		Get.InputField.r_ApparentPhasePower[Phases.L1]:= r_ApparentPower[Phases.L1];
		Get.InputField.r_ApparentPhasePower[Phases.L2]:= r_ApparentPower[Phases.L2];
		Get.InputField.r_ApparentPhasePower[Phases.L3]:= r_ApparentPower[Phases.L3];		
		Get.InputField.r_ApparentPhasePower[Phases.AVG]:= (r_ApparentPower[Phases.L1] + r_ApparentPower[Phases.L2] + r_ApparentPower[Phases.L3]);	
		Get.InputField.r_ApparentPower := r_ApparentPower[Phases.L1]+ r_ApparentPower[Phases.L2] + r_ApparentPower[Phases.L3];
		
		Get.InputField.r_ReactivePhasePower[Phases.L1]:= r_ReactivePower[Phases.L1];
		Get.InputField.r_ReactivePhasePower[Phases.L2]:= r_ReactivePower[Phases.L2];
		Get.InputField.r_ReactivePhasePower[Phases.L3]:= r_ReactivePower[Phases.L3];		
		Get.InputField.r_ReactivePhasePower[Phases.AVG]:= (r_ReactivePower[Phases.L1] + r_ReactivePower[Phases.L2] + r_ReactivePower[Phases.L3]);	
		Get.InputField.r_ReactivePower := r_ReactivePower[Phases.L1]+ r_ReactivePower[Phases.L2] + r_ReactivePower[Phases.L3];
		
		//Energy Consumed                           
		Get.InputField.r_EnergyConsumed		 :=		LINT_TO_REAL(r_ActiveEnergyNegative);	
	                                                
		//Energy Delivered                          
		Get.InputField.r_EnergySupplied :=		LINT_TO_REAL(r_ActiveEnergyPositive);		
	    
		//Powerfactors                                                                 
	    Get.InputField.r_PowerFactor[Phases.L1]:= r_PowerFactor[Phases.L1];
		Get.InputField.r_PowerFactor[Phases.L2]:= r_PowerFactor[Phases.L2];
		Get.InputField.r_PowerFactor[Phases.L3]:= r_PowerFactor[Phases.L3];		
		Get.InputField.r_PowerFactor[Phases.AVG]:= (r_PowerFactor[Phases.L1] + r_PowerFactor[Phases.L2] + r_PowerFactor[Phases.L3])/3;	                                            

		//THD not in EL3443                                                       
		//VoltageUnbalance  not in EL3443   
		
		//EL3443 only gives a boolean for fieldRotation with True meaning right.
		//So false could be none or left. Check voltages before checking rotation.
		IF (Get.InputField.r_LineVoltage[Phases.L1] > 300) AND (Get.InputField.r_LineVoltage[Phases.L2] > 300) AND (Get.InputField.r_LineVoltage[Phases.L3] > 300) THEN
			IF  TotalStatus.bit_GridDirection THEN
				Get.InputField.e_ACrotationStatus := eACRotationState.Right;
			ELSE
				Get.InputField.e_ACrotationStatus := eACRotationState.Left;	
			END_IF
		ELSE
			Get.InputField.e_ACrotationStatus := eACRotationState.None;	
		END_IF
		get.events.b_EL3443Warning := FALSE;
		EL3443FaultCounter := 0;
		
	ELSE
		//faultwarning sets directly if the card states an error.
		//Fault error only sets if the fault remains for a longer period of time.
		get.events.b_EL3443Warning := TRUE;
		EL3443FaultCounter := EL3443FaultCounter +1;
		IF EL3443FaultCounter > 50 THEN
			get.events.b_EL3443Error := TRUE;
		END_IF
	END_IF
END_IF

END_FUNCTION_BLOCK

// ---- POUs/Objects/PowerQualityMonitor/FB_Janitza_UMG801/FB_Janitza.TcPOU
FUNCTION_BLOCK FB_Janitza
VAR_IN_OUT
	get					: ST_PowerMonitor_get;
END_VAR
VAR
	MBRead: FB_MBReadRegs;
	w_MBStartAddress	:	WORD;
	//Set 1 is bigger, as this includes voltage measurements.
	DataBuffer		: 	ARRAY[0..62] OF REAL;
	SecondDataBuffer		: 	ARRAY[0..62] OF REAL;
	tempword	:	dword;	
	temp	:	BOOL;
	UI_Iterator	:	UINT;
	//retrieve new data every 100ms
	GetDataTimer	:	TON := (PT := TIME#100MS);
END_VAR

VAR_INPUT
	ReadData: BOOL;
	b_TNmodeEnable		AT %Q* : BOOL;
END_VAR

VAR
	ast_InputPowerlockData	:	ARRAY[1..2] OF ST_Powerlockdata;
	ast_OutputPowerlockData	:	ARRAY[1..3] OF ST_Powerlockdata;

	StartTransmissionEdge : R_Trig;
	TransmissionDone	:	F_trig;
	
	ui_MBRetryCount	:	uint;
	
	b_busy: BOOL;
	b_CommError: BOOL;
	udi_errid: UDINT;
	udi_cbread: UDINT;
	
	testWord	:	DWORD;
	testWordB	:	WORD;
	testWordC	:	WORD;
END_VAR



//While ReadData is true, initiate data transfer every 100ms;
GetDataTimer(in:= ((NOT GetDataTimer.Q) AND ReadData));

//ReadJanitzaData();
ReadDataSFC();

ACTION aCombineInputData:
IF PowerMeterConfig.b_InputFieldsAvailable THEN
	//Combine shared data from output fields into get struct
	get.InputField.r_Current[Phases.L1] :=	get.InputField.ar_PowerlockCurrents[1][Phases.L1] + 
											get.InputField.ar_PowerlockCurrents[2][Phases.L1];
	
	get.InputField.r_Current[Phases.L2] :=	get.InputField.ar_PowerlockCurrents[1][Phases.L2] + 
											get.InputField.ar_PowerlockCurrents[2][Phases.L2];
	
	get.InputField.r_Current[Phases.L3] :=	get.InputField.ar_PowerlockCurrents[1][Phases.L3] + 
											get.InputField.ar_PowerlockCurrents[2][Phases.L3];			
	
	get.InputField.r_Current[Phases.N] :=	get.InputField.ar_PowerlockCurrents[1][Phases.N] + 
											get.InputField.ar_PowerlockCurrents[2][Phases.N];			
	
	get.InputField.r_Current[Phases.AVG] :=	(get.InputField.r_Current[Phases.L1] + 
											get.InputField.r_Current[Phases.L2] +
											get.InputField.r_Current[Phases.L3])/3;							
	
	Get.InputField.r_ActivePhasePower[Phases.L1]	:=	ast_InputPowerLockData[1].r_ActivePhasePower[Phases.L1] + 
														ast_InputPowerLockData[2].r_ActivePhasePower[Phases.L1];
	
	Get.InputField.r_ActivePhasePower[Phases.L2]	:=	ast_InputPowerLockData[1].r_ActivePhasePower[Phases.L2] + 
														ast_InputPowerLockData[2].r_ActivePhasePower[Phases.L2];
														
	Get.InputField.r_ActivePhasePower[Phases.L3]	:=	ast_InputPowerLockData[1].r_ActivePhasePower[Phases.L3] + 
														ast_InputPowerLockData[2].r_ActivePhasePower[Phases.L3];
														
	Get.InputField.r_ActivePhasePower[Phases.AVG]	:=	ast_InputPowerLockData[1].r_ActivePhasePower[Phases.AVG] + 
														ast_InputPowerLockData[2].r_ActivePhasePower[Phases.AVG];									
	
														
														
	Get.InputField.r_ApparentPhasePower[Phases.L1]	:=	ast_InputPowerLockData[1].r_ApparentPhasePower[Phases.L1] + 
														ast_InputPowerLockData[2].r_ApparentPhasePower[Phases.L1];
	
	Get.InputField.r_ApparentPhasePower[Phases.L2]	:=	ast_InputPowerLockData[1].r_ApparentPhasePower[Phases.L2] + 
														ast_InputPowerLockData[2].r_ApparentPhasePower[Phases.L2];
														
	Get.InputField.r_ApparentPhasePower[Phases.L3]	:=	ast_InputPowerLockData[1].r_ApparentPhasePower[Phases.L3] + 
														ast_InputPowerLockData[2].r_ApparentPhasePower[Phases.L3];
														
	Get.InputField.r_ApparentPhasePower[Phases.AVG]	:=	ast_InputPowerLockData[1].r_ApparentPhasePower[Phases.AVG] + 
														ast_InputPowerLockData[2].r_ApparentPhasePower[Phases.AVG];	

														
														
	Get.InputField.r_ReactivePhasePower[Phases.L1]	:=	ast_InputPowerLockData[1].r_ReactivePhasePower[Phases.L1] + 
														ast_InputPowerLockData[2].r_ReactivePhasePower[Phases.L1];
	
	Get.InputField.r_ReactivePhasePower[Phases.L2]	:=	ast_InputPowerLockData[1].r_ReactivePhasePower[Phases.L2] + 
														ast_InputPowerLockData[2].r_ReactivePhasePower[Phases.L2];
														
	Get.InputField.r_ReactivePhasePower[Phases.L3]	:=	ast_InputPowerLockData[1].r_ReactivePhasePower[Phases.L3] + 
														ast_InputPowerLockData[2].r_ReactivePhasePower[Phases.L3];
														
	Get.InputField.r_ReactivePhasePower[Phases.AVG]	:=	ast_InputPowerLockData[1].r_ReactivePhasePower[Phases.AVG] + 
														ast_InputPowerLockData[2].r_ReactivePhasePower[Phases.AVG];	


										
	Get.InputField.r_ActivePower		:=	ast_InputPowerLockData[1].r_ActivePower + 
											ast_InputPowerLockData[2].r_ActivePower;
	
	Get.InputField.r_ApparentPower		:=	ast_InputPowerLockData[1].r_ApparentPower + 
											ast_InputPowerLockData[2].r_ApparentPower;
											
	Get.InputField.r_ReactivePower		:=	ast_InputPowerLockData[1].r_ReactivePower + 
											ast_InputPowerLockData[2].r_ReactivePower;
	
	Get.InputField.r_EnergyConsumed		:=	ast_InputPowerLockData[1].r_EnergyConsumed + 
											ast_InputPowerLockData[2].r_EnergyConsumed;
	
	Get.InputField.r_EnergySupplied		:=	ast_InputPowerLockData[1].r_EnergySupplied + 
											ast_InputPowerLockData[2].r_EnergySupplied;
	
	get.InputField.r_PowerFactor[Phases.L1] :=		(ast_InputPowerLockData[1].ar_PowerFactor[Phases.L1] + 
													ast_InputPowerLockData[2].ar_PowerFactor[Phases.L1] )/2;	
														
	get.InputField.r_PowerFactor[Phases.L2] :=		(ast_InputPowerLockData[1].ar_PowerFactor[Phases.L2] + 
													ast_InputPowerLockData[2].ar_PowerFactor[Phases.L2])/2;		
	
	get.InputField.r_PowerFactor[Phases.L3] :=		(ast_InputPowerLockData[1].ar_PowerFactor[Phases.L3] + 
													ast_InputPowerLockData[2].ar_PowerFactor[Phases.L3])/2;
	
	get.InputField.r_THD[Phases.L1] 		:=		(ast_InputPowerLockData[1].ar_THD[Phases.L1] + 
													ast_InputPowerLockData[2].ar_THD[Phases.L1])/2;
														
	get.InputField.r_THD[Phases.L2] 		:=		(ast_InputPowerLockData[1].ar_THD[Phases.L2] + 
													ast_InputPowerLockData[2].ar_THD[Phases.L2])/2;	
	
	get.InputField.r_THD[Phases.L3]		 	:=		(ast_InputPowerLockData[1].ar_THD[Phases.L3] + 
													ast_InputPowerLockData[2].ar_THD[Phases.L3])/2;											
	
	get.InputField.r_PowerFactor[Phases.AVG] :=	(get.InputField.r_PowerFactor[Phases.L1] + 
													get.InputField.r_PowerFactor[Phases.L2] + 
													get.InputField.r_PowerFactor[Phases.L3])/3;		
	
	get.InputField.r_THD[Phases.AVG] :=			(get.InputField.r_THD[Phases.L1] + 
													get.InputField.r_THD[Phases.L2] + 
													get.InputField.r_THD[Phases.L3])/3;
end_if
END_ACTION

ACTION aCombineOutputData:

//Combine shared data from output fields into get struct
get.OutputField.r_Current[Phases.L1] :=	get.OutputField.ar_PowerlockCurrents[1][Phases.L1] + 
										get.OutputField.ar_PowerlockCurrents[2][Phases.L1] + 
										get.OutputField.ar_PowerlockCurrents[3][Phases.L1];

get.OutputField.r_Current[Phases.L2] :=	get.OutputField.ar_PowerlockCurrents[1][Phases.L2] + 
										get.OutputField.ar_PowerlockCurrents[2][Phases.L2] + 
										get.OutputField.ar_PowerlockCurrents[3][Phases.L2];

get.OutputField.r_Current[Phases.L3] :=	get.OutputField.ar_PowerlockCurrents[1][Phases.L3] + 
										get.OutputField.ar_PowerlockCurrents[2][Phases.L3] + 
										get.OutputField.ar_PowerlockCurrents[3][Phases.L3];			

get.OutputField.r_Current[Phases.N] :=	get.OutputField.ar_PowerlockCurrents[1][Phases.N] + 
										get.OutputField.ar_PowerlockCurrents[2][Phases.N] + 
										get.OutputField.ar_PowerlockCurrents[3][Phases.N];			

get.OutputField.r_Current[Phases.AVG] :=	(get.OutputField.r_Current[Phases.L1] + 
											get.OutputField.r_Current[Phases.L2] +
											get.OutputField.r_Current[Phases.L3])/3;							

Get.OutputField.r_ActivePhasePower[Phases.L1]	:=	ast_OutputPowerLockData[1].r_ActivePhasePower[Phases.L1] + 
													ast_OutputPowerLockData[2].r_ActivePhasePower[Phases.L1] +
													ast_OutputPowerLockData[3].r_ActivePhasePower[Phases.L1];
	
Get.OutputField.r_ActivePhasePower[Phases.L2]	:=	ast_OutputPowerLockData[1].r_ActivePhasePower[Phases.L2] + 
													ast_OutputPowerLockData[2].r_ActivePhasePower[Phases.L2] +
													ast_OutputPowerLockData[3].r_ActivePhasePower[Phases.L2];
														
Get.OutputField.r_ActivePhasePower[Phases.L3]	:=	ast_OutputPowerLockData[1].r_ActivePhasePower[Phases.L3] + 
													ast_OutputPowerLockData[2].r_ActivePhasePower[Phases.L3] + 
													ast_OutputPowerLockData[3].r_ActivePhasePower[Phases.L3];
														
Get.OutputField.r_ActivePhasePower[Phases.AVG]	:=	ast_OutputPowerLockData[1].r_ActivePhasePower[Phases.AVG] + 
													ast_OutputPowerLockData[2].r_ActivePhasePower[Phases.AVG] +
													ast_OutputPowerLockData[3].r_ActivePhasePower[Phases.AVG];									
	
														
														
Get.OutputField.r_ApparentPhasePower[Phases.L1]	:=	ast_OutputPowerLockData[1].r_ApparentPhasePower[Phases.L1] + 
													ast_OutputPowerLockData[2].r_ApparentPhasePower[Phases.L1] +
													ast_OutputPowerLockData[3].r_ApparentPhasePower[Phases.L1];
	
Get.OutputField.r_ApparentPhasePower[Phases.L2]	:=	ast_OutputPowerLockData[1].r_ApparentPhasePower[Phases.L2] + 
													ast_OutputPowerLockData[2].r_ApparentPhasePower[Phases.L2] +
													ast_OutputPowerLockData[3].r_ApparentPhasePower[Phases.L2];
														
Get.OutputField.r_ApparentPhasePower[Phases.L3]	:=	ast_OutputPowerLockData[1].r_ApparentPhasePower[Phases.L3] + 
													ast_OutputPowerLockData[2].r_ApparentPhasePower[Phases.L3] +
													ast_OutputPowerLockData[3].r_ApparentPhasePower[Phases.L3];
														
Get.OutputField.r_ApparentPhasePower[Phases.AVG]:=	ast_OutputPowerLockData[1].r_ApparentPhasePower[Phases.AVG] + 
													ast_OutputPowerLockData[2].r_ApparentPhasePower[Phases.AVG] +
													ast_OutputPowerLockData[3].r_ApparentPhasePower[Phases.AVG];	
														
													
													
Get.OutputField.r_ReactivePhasePower[Phases.L1]	:=	ast_OutputPowerLockData[1].r_ReactivePhasePower[Phases.L1] + 
													ast_OutputPowerLockData[2].r_ReactivePhasePower[Phases.L1] +
													ast_OutputPowerLockData[3].r_ReactivePhasePower[Phases.L1];	
	
Get.OutputField.r_ReactivePhasePower[Phases.L2]	:=	ast_OutputPowerLockData[1].r_ReactivePhasePower[Phases.L2] + 
													ast_OutputPowerLockData[2].r_ReactivePhasePower[Phases.L2] +
													ast_OutputPowerLockData[3].r_ReactivePhasePower[Phases.L2];	
														
Get.OutputField.r_ReactivePhasePower[Phases.L3]	:=	ast_OutputPowerLockData[1].r_ReactivePhasePower[Phases.L3] + 
													ast_OutputPowerLockData[2].r_ReactivePhasePower[Phases.L3] +
													ast_OutputPowerLockData[3].r_ReactivePhasePower[Phases.L3];	
														
Get.OutputField.r_ReactivePhasePower[Phases.AVG]:=	ast_OutputPowerLockData[1].r_ReactivePhasePower[Phases.AVG] + 
													ast_OutputPowerLockData[2].r_ReactivePhasePower[Phases.AVG] +	
													ast_OutputPowerLockData[3].r_ReactivePhasePower[Phases.AVG];												
											
											
Get.OutputField.r_ActivePower		:=	ast_OutputPowerLockData[1].r_ActivePower + 
										ast_OutputPowerLockData[2].r_ActivePower + 
										ast_OutputPowerLockData[3].r_ActivePower;

Get.OutputField.r_ApparentPower		:=	ast_OutputPowerLockData[1].r_ApparentPower + 
										ast_OutputPowerLockData[2].r_ApparentPower + 
										ast_OutputPowerLockData[3].r_ApparentPower;

Get.OutputField.r_ReactivePower		:=	ast_OutputPowerLockData[1].r_ReactivePower + 
										ast_OutputPowerLockData[2].r_ReactivePower + 
										ast_OutputPowerLockData[3].r_ReactivePower;

Get.OutputField.r_EnergyConsumed	:=	ast_OutputPowerLockData[1].r_EnergyConsumed + 
										ast_OutputPowerLockData[2].r_EnergyConsumed + 
										ast_OutputPowerLockData[3].r_EnergyConsumed;

Get.OutputField.r_EnergySupplied	:=	ast_OutputPowerLockData[1].r_EnergySupplied + 
										ast_OutputPowerLockData[2].r_EnergySupplied + 
										ast_OutputPowerLockData[3].r_EnergySupplied;

//if 3 output fields are available, calculate averages over 3 fields. Otherwise over 2
IF PowerMeterConfig.b_ThirdOutputFieldAvailable THEN
	get.OutputField.r_PowerFactor[Phases.L1] :=		(ast_OutputPowerLockData[1].ar_PowerFactor[Phases.L1] + 
													ast_OutputPowerLockData[2].ar_PowerFactor[Phases.L1] + 
													ast_OutputPowerLockData[3].ar_PowerFactor[Phases.L1])/3;	
													
	get.OutputField.r_PowerFactor[Phases.L2] :=		(ast_OutputPowerLockData[1].ar_PowerFactor[Phases.L2] + 
													ast_OutputPowerLockData[2].ar_PowerFactor[Phases.L2] + 
													ast_OutputPowerLockData[3].ar_PowerFactor[Phases.L2])/3;		

	get.OutputField.r_PowerFactor[Phases.L3] :=		(ast_OutputPowerLockData[1].ar_PowerFactor[Phases.L3] + 
													ast_OutputPowerLockData[2].ar_PowerFactor[Phases.L3] + 
													ast_OutputPowerLockData[3].ar_PowerFactor[Phases.L3])/3;	

	get.OutputField.r_THD[Phases.L1] 		:=		(ast_OutputPowerLockData[1].ar_THD[Phases.L1] + 
													ast_OutputPowerLockData[2].ar_THD[Phases.L1] + 
													ast_OutputPowerLockData[3].ar_THD[Phases.L1])/3;	
													
	get.OutputField.r_THD[Phases.L2] 		:=		(ast_OutputPowerLockData[1].ar_THD[Phases.L2] + 
													ast_OutputPowerLockData[2].ar_THD[Phases.L2] + 
													ast_OutputPowerLockData[3].ar_THD[Phases.L2])/3;		

	get.OutputField.r_THD[Phases.L3]		 :=		(ast_OutputPowerLockData[1].ar_THD[Phases.L3] + 
													ast_OutputPowerLockData[2].ar_THD[Phases.L3] + 
													ast_OutputPowerLockData[3].ar_THD[Phases.L3])/3;														
ELSE
	get.OutputField.r_PowerFactor[Phases.L1] :=		(ast_OutputPowerLockData[1].ar_PowerFactor[Phases.L1] + 
													ast_OutputPowerLockData[2].ar_PowerFactor[Phases.L1] )/2;	
													
	get.OutputField.r_PowerFactor[Phases.L2] :=		(ast_OutputPowerLockData[1].ar_PowerFactor[Phases.L2] + 
													ast_OutputPowerLockData[2].ar_PowerFactor[Phases.L2])/2;		

	get.OutputField.r_PowerFactor[Phases.L3] :=		(ast_OutputPowerLockData[1].ar_PowerFactor[Phases.L3] + 
													ast_OutputPowerLockData[2].ar_PowerFactor[Phases.L3])/2;

	get.OutputField.r_THD[Phases.L1] 		:=		(ast_OutputPowerLockData[1].ar_THD[Phases.L1] + 
													ast_OutputPowerLockData[2].ar_THD[Phases.L1])/2;
													
	get.OutputField.r_THD[Phases.L2] 		:=		(ast_OutputPowerLockData[1].ar_THD[Phases.L2] + 
													ast_OutputPowerLockData[2].ar_THD[Phases.L2])/2;	

	get.OutputField.r_THD[Phases.L3]		 :=		(ast_OutputPowerLockData[1].ar_THD[Phases.L3] + 
													ast_OutputPowerLockData[2].ar_THD[Phases.L3])/2;											
END_IF



get.OutputField.r_PowerFactor[Phases.AVG] :=	(get.OutputField.r_PowerFactor[Phases.L1] + 
												get.OutputField.r_PowerFactor[Phases.L2] + 
												get.OutputField.r_PowerFactor[Phases.L3])/3;		

get.OutputField.r_THD[Phases.AVG] :=			(get.OutputField.r_THD[Phases.L1] + 
												get.OutputField.r_THD[Phases.L2] + 
												get.OutputField.r_THD[Phases.L3])/3;
END_ACTION

ACTION aReadInputField1:

IF NOT PowerMeterConfig.b_InputFieldsAvailable THEN
	//skip this step if input fields are not in use
	SFCTip := TRUE;
ELSE
	
	IF PowerMeterconfig.b_ThirdOutputFieldAvailable THEN
		//if third output field is available, Input field is connected to module 2, so inputfield 1 is address 19600
		w_MBStartAddress := 19600;
	ELSE
		//if no third output field is available, Input field is connected to module 1, so inputfield 1 is address 19400
		w_MBStartAddress := 19400;
	END_IF

	MBRead(
	sIPAddr := PowerMeterConfig.IP_JANITZA,
	nTCPPort := PowerMeterConfig.MBPort_Janitza,
	nUnitID := 1,//16#FF;
	nMBAddr := w_MBStartAddress,
	nQuantity := 50*2,
	cbLength := SIZEOF(DataBuffer),
	pDestAddr := ADR(DataBuffer),
	bExecute := NOT (b_busy OR TransmissionDone.Q),	//	<- werkt dit niet gewoon?
	bBusy => b_busy,
	bError => b_CommError,
	nErrId => udi_errid,
	cbRead => udi_cbread,
	tTimeout := T#25MS
	);
	
	TransmissionDone(clk := b_busy);
	
	IF TransmissionDone.q THEN
		IF NOT b_CommError  THEN	
			
			FOR UI_Iterator := 0 TO 50 BY 1 DO
				DataBuffer[UI_Iterator] := ChangeRealEndianess(DataBuffer[UI_Iterator]);
			END_FOR 
			//field specific data, keep separate at first. Then combine data into get struct in a later step.
			get.InputField.ar_PowerlockCurrents[1][Phases.L1] := DataBuffer[0];
			get.InputField.ar_PowerlockCurrents[1][Phases.L2] := DataBuffer[1];
			get.InputField.ar_PowerlockCurrents[1][Phases.L3] := DataBuffer[2];
			get.InputField.ar_PowerlockCurrents[1][Phases.N] := DataBuffer[3];
			
			ast_InputPowerLockData[1].r_ActivePhasePower[phases.L1] := DataBuffer[4];
       		ast_InputPowerLockData[1].r_ActivePhasePower[phases.L2] := DataBuffer[5];
			ast_InputPowerLockData[1].r_ActivePhasePower[phases.L3] := DataBuffer[6];
			ast_InputPowerLockData[1].r_ActivePhasePower[phases.AVG] := (DataBuffer[4] + DataBuffer[5] + DataBuffer[6])/3;
		    
			ast_InputPowerLockData[1].r_ApparentPhasePower[phases.L1] := DataBuffer[8];
       		ast_InputPowerLockData[1].r_ApparentPhasePower[phases.L2] := DataBuffer[9];
			ast_InputPowerLockData[1].r_ApparentPhasePower[phases.L3] := DataBuffer[10];
			ast_InputPowerLockData[1].r_ApparentPhasePower[phases.AVG] := (DataBuffer[8] + DataBuffer[9] + DataBuffer[10])/3;
		    
			ast_InputPowerLockData[1].r_ReactivePhasePower[phases.L1] := DataBuffer[12];
       		ast_InputPowerLockData[1].r_ReactivePhasePower[phases.L2] := DataBuffer[13];
			ast_InputPowerLockData[1].r_ReactivePhasePower[phases.L3] := DataBuffer[14];
			ast_InputPowerLockData[1].r_ReactivePhasePower[phases.AVG] := (DataBuffer[12] + DataBuffer[13] + DataBuffer[14])/3;
		    
			ast_InputPowerLockData[1].r_ActivePower := DataBuffer[7];
			ast_InputPowerLockData[1].r_ApparentPower := DataBuffer[11];
			ast_InputPowerLockData[1].r_ReactivePower := DataBuffer[15];
					               
			ast_InputPowerLockData[1].ar_PowerFactor[Phases.L1] := DataBuffer[16];
			ast_InputPowerLockData[1].ar_PowerFactor[Phases.L2] := DataBuffer[17];
			ast_InputPowerLockData[1].ar_PowerFactor[Phases.L3] := DataBuffer[18];
			ast_InputPowerLockData[1].ar_PowerFactor[Phases.AVG] := (DataBuffer[16] + DataBuffer[17] + DataBuffer[18])/3;
					               
			ast_InputPowerLockData[1].r_EnergyConsumed	:=  DataBuffer[26];
			ast_InputPowerLockData[1].r_EnergySupplied 	:=	DataBuffer[30];
					               
			ast_InputPowerLockData[1].ar_THD[Phases.L1] := DataBuffer[47];
			ast_InputPowerLockData[1].ar_THD[Phases.L2] := DataBuffer[48];
			ast_InputPowerLockData[1].ar_THD[Phases.L3] := DataBuffer[49];
				
			ui_MBRetryCount := 0;
			sfctip := TRUE;
		ELSE
			ui_MBRetryCount := ui_MBRetryCount + 1;
			
			IF ui_MBRetryCount > 1 THEN
				get.events.b_MBCommWarning := TRUE;
			END_IF	
			
			//if comm fails 5 times in a row. try next input
			IF ui_MBRetryCount > 4 THEN
				get.Events.b_MBCommError := TRUE;
				sfctip := TRUE;
			END_IF
		END_IF
	END_IF
END_IF
END_ACTION

ACTION aReadInputField2:

IF NOT PowerMeterConfig.b_InputFieldsAvailable THEN
	//skip this step if input fields are not in use
	SFCTip := TRUE;
ELSE
	
	IF PowerMeterconfig.b_ThirdOutputFieldAvailable THEN
		//if third output field is available, Input field is connected to module 2, so inputfield 2 is address 19700
		w_MBStartAddress := 19700;
	ELSE
		//if no third output field is available, Input field is connected to module 1, so inputfield 2 is address 19500
		w_MBStartAddress := 19500;
	END_IF

	MBRead(
	sIPAddr := PowerMeterConfig.IP_JANITZA,
	nTCPPort := PowerMeterConfig.MBPort_Janitza,
	nUnitID := 1,//16#FF;
	nMBAddr := w_MBStartAddress,
	nQuantity := 50*2,
	cbLength := SIZEOF(DataBuffer),
	pDestAddr := ADR(DataBuffer),
	bExecute := NOT (b_busy OR TransmissionDone.Q),	//	<- werkt dit niet gewoon?
	bBusy => b_busy,
	bError => b_CommError,
	nErrId => udi_errid,
	cbRead => udi_cbread,
	tTimeout := T#25MS
	);
	
	TransmissionDone(clk := b_busy);
	
	IF TransmissionDone.q THEN
		IF NOT b_CommError THEN	
			
			FOR UI_Iterator := 0 TO 50 BY 1 DO
				DataBuffer[UI_Iterator] := ChangeRealEndianess(DataBuffer[UI_Iterator]);
			END_FOR 
			
			//field specific data, keep separate at first. Then combine data into get struct in a later step.
			get.InputField.ar_PowerlockCurrents[2][Phases.L1] := DataBuffer[0];
			get.InputField.ar_PowerlockCurrents[2][Phases.L2] := DataBuffer[1];
			get.InputField.ar_PowerlockCurrents[2][Phases.L3] := DataBuffer[2];
			get.InputField.ar_PowerlockCurrents[2][Phases.N] := DataBuffer[3];
			
			ast_InputPowerLockData[2].r_ActivePhasePower[phases.L1] := DataBuffer[4];
       		ast_InputPowerLockData[2].r_ActivePhasePower[phases.L2] := DataBuffer[5];
			ast_InputPowerLockData[2].r_ActivePhasePower[phases.L3] := DataBuffer[6];
			ast_InputPowerLockData[2].r_ActivePhasePower[phases.AVG] := (DataBuffer[4] + DataBuffer[5] + DataBuffer[6])/3;
		                           
			ast_InputPowerLockData[2].r_ApparentPhasePower[phases.L1] := DataBuffer[8];
       		ast_InputPowerLockData[2].r_ApparentPhasePower[phases.L2] := DataBuffer[9];
			ast_InputPowerLockData[2].r_ApparentPhasePower[phases.L3] := DataBuffer[10];
			ast_InputPowerLockData[2].r_ApparentPhasePower[phases.AVG] := (DataBuffer[8] + DataBuffer[9] + DataBuffer[10])/3;
		                           
			ast_InputPowerLockData[2].r_ReactivePhasePower[phases.L1] := DataBuffer[12];
       		ast_InputPowerLockData[2].r_ReactivePhasePower[phases.L2] := DataBuffer[13];
			ast_InputPowerLockData[2].r_ReactivePhasePower[phases.L3] := DataBuffer[14];
			ast_InputPowerLockData[2].r_ReactivePhasePower[phases.AVG] := (DataBuffer[12] + DataBuffer[13] + DataBuffer[14])/3;
		    			
			ast_InputPowerLockData[2].r_ActivePower := DataBuffer[7];
			ast_InputPowerLockData[2].r_ApparentPower := DataBuffer[11];
			ast_InputPowerLockData[2].r_ReactivePower := DataBuffer[15];
					               
			ast_InputPowerLockData[2].ar_PowerFactor[Phases.L1] := DataBuffer[16];
			ast_InputPowerLockData[2].ar_PowerFactor[Phases.L2] := DataBuffer[17];
			ast_InputPowerLockData[2].ar_PowerFactor[Phases.L3] := DataBuffer[18];
			ast_InputPowerLockData[2].ar_PowerFactor[Phases.AVG] := (DataBuffer[16] + DataBuffer[17] + DataBuffer[18])/3;
					               
			ast_InputPowerLockData[2].r_EnergyConsumed	:=  DataBuffer[26];
			ast_InputPowerLockData[2].r_EnergySupplied 	:=	DataBuffer[30];
					               
			ast_InputPowerLockData[2].ar_THD[Phases.L1] := DataBuffer[47];
			ast_InputPowerLockData[2].ar_THD[Phases.L2] := DataBuffer[48];
			ast_InputPowerLockData[2].ar_THD[Phases.L3] := DataBuffer[49];
				
			ui_MBRetryCount := 0;
			sfctip := TRUE;
		ELSE
			ui_MBRetryCount := ui_MBRetryCount + 1;
			
			
			IF ui_MBRetryCount > 1 THEN
				get.events.b_MBCommWarning := TRUE;
			END_IF	
			
			//if comm fails 5 times in a row. try next input
			IF ui_MBRetryCount > 4 THEN
				get.Events.b_MBCommError := TRUE;
				sfctip := TRUE;
			END_IF
		END_IF
	END_IF
END_IF
END_ACTION

ACTION aReadInternalField:

MBRead(
sIPAddr := PowerMeterConfig.IP_JANITZA,
nTCPPort := PowerMeterConfig.MBPort_Janitza,
nUnitID := 1,//16#FF;
nMBAddr := 19300,
nQuantity := 50*2,
cbLength := SIZEOF(DataBuffer),
pDestAddr := ADR(DataBuffer),
bExecute := NOT (b_busy OR TransmissionDone.Q),	//	<- werkt dit niet gewoon?
bBusy => b_busy,
bError => b_CommError,
nErrId => udi_errid,
cbRead => udi_cbread,
tTimeout := T#25MS
);

TransmissionDone(clk := b_busy);

IF TransmissionDone.q THEN
	IF NOT b_CommError  THEN	
		
		FOR UI_Iterator := 0 TO 50 BY 1 DO
			DataBuffer[UI_Iterator] := ChangeRealEndianess(DataBuffer[UI_Iterator]);
		END_FOR 
		
		//field specific data, keep separate at first. Then combine data into get struct in a later step.
		get.InternalSupply.r_Current[Phases.L1] := DataBuffer[0];
		get.InternalSupply.r_Current[Phases.L2] := DataBuffer[1];
		get.InternalSupply.r_Current[Phases.L3] := DataBuffer[2];
		get.InternalSupply.r_Current[Phases.N] := DataBuffer[3];
		get.InternalSupply.r_Current[Phases.AVG] := (DataBuffer[0] + DataBuffer[1] + DataBuffer[2])/3;
		
		get.InternalSupply.r_ActivePhasePower[phases.L1] := DataBuffer[4];
   		get.InternalSupply.r_ActivePhasePower[phases.L2] := DataBuffer[5];
		get.InternalSupply.r_ActivePhasePower[phases.L3] := DataBuffer[6];
		get.InternalSupply.r_ActivePhasePower[phases.AVG] := (DataBuffer[4] + DataBuffer[5] + DataBuffer[6])/3;
		
		get.InternalSupply.r_ApparentPhasePower[phases.L1] := DataBuffer[8];
   		get.InternalSupply.r_ApparentPhasePower[phases.L2] := DataBuffer[9];
		get.InternalSupply.r_ApparentPhasePower[phases.L3] := DataBuffer[10];
		get.InternalSupply.r_ApparentPhasePower[phases.AVG] := (DataBuffer[8] + DataBuffer[9] + DataBuffer[10])/3;
		
		get.InternalSupply.r_ReactivePhasePower[phases.L1] := DataBuffer[12];
   		get.InternalSupply.r_ReactivePhasePower[phases.L2] := DataBuffer[13];
		get.InternalSupply.r_ReactivePhasePower[phases.L3] := DataBuffer[14];
		get.InternalSupply.r_ReactivePhasePower[phases.AVG] := (DataBuffer[12] + DataBuffer[13] + DataBuffer[14])/3;
		    				                        
		get.InternalSupply.r_ActivePower := DataBuffer[7];
		get.InternalSupply.r_ApparentPower := DataBuffer[11];
		get.InternalSupply.r_ReactivePower := DataBuffer[15];
        
		get.InternalSupply.r_PowerFactor[Phases.L1] := DataBuffer[16];
		get.InternalSupply.r_PowerFactor[Phases.L2] := DataBuffer[17];
		get.InternalSupply.r_PowerFactor[Phases.L3] := DataBuffer[18];
		get.InternalSupply.r_PowerFactor[Phases.AVG] := (DataBuffer[16] + DataBuffer[17] + DataBuffer[18])/3;
		
		get.InternalSupply.r_EnergyConsumed	:=  DataBuffer[26];
		get.InternalSupply.r_EnergySupplied 	:=	DataBuffer[30];
		
		get.InternalSupply.r_THD[Phases.L1] := DataBuffer[47];
		get.InternalSupply.r_THD[Phases.L2] := DataBuffer[48];
		get.InternalSupply.r_THD[Phases.L3] := DataBuffer[49];
			
		ui_MBRetryCount := 0;
		sfctip := TRUE;
	ELSE
		ui_MBRetryCount := ui_MBRetryCount + 1;
				
		IF ui_MBRetryCount > 1 THEN
			get.events.b_MBCommWarning := TRUE;
		END_IF	
		
		//if comm fails 5 times in a row. try next input
		IF ui_MBRetryCount > 4 THEN
			get.Events.b_MBCommError := TRUE;
			sfctip := TRUE;
		END_IF
	END_IF
END_IF
END_ACTION

ACTION aReadOutputField1:

MBRead(
sIPAddr := PowerMeterConfig.IP_JANITZA,
nTCPPort := PowerMeterConfig.MBPort_Janitza,
nUnitID := 1,
nMBAddr := 19000,
nQuantity := 61*2,
cbLength := SIZEOF(DataBuffer),
pDestAddr := ADR(DataBuffer),
bExecute := NOT (b_busy OR TransmissionDone.Q),	//	<- werkt dit niet gewoon?
bBusy => b_busy,
bError => b_CommError,
nErrId => udi_errid,
cbRead => udi_cbread,
tTimeout := T#25MS
);

TransmissionDone(clk := b_busy);

IF TransmissionDone.q THEN
	Temp := FALSE;
	IF NOT b_CommError then
		//General inputfield data, can be pushed to get struct immediately
		
		FOR UI_Iterator := 0 TO 61 BY 1 DO
			DataBuffer[UI_Iterator] := ChangeRealEndianess(DataBuffer[UI_Iterator]);
		END_FOR 
		
		get.OutputField.r_PhaseVoltage[Phases.L1] := DataBuffer[0];
		get.OutputField.r_PhaseVoltage[Phases.L2] := DataBuffer[1];
		get.OutputField.r_PhaseVoltage[Phases.L3] := DataBuffer[2];
		get.OutputField.r_PhaseVoltage[Phases.AVG] := (DataBuffer[0]+DataBuffer[1]+DataBuffer[2])/3;
		
		get.OutputField.r_LineVoltage[Phases.L1] := DataBuffer[3];
		get.OutputField.r_LineVoltage[Phases.L2] := DataBuffer[4];
		get.OutputField.r_LineVoltage[Phases.L3] := DataBuffer[5];
		get.OutputField.r_LineVoltage[Phases.AVG] := (DataBuffer[3]+DataBuffer[4]+DataBuffer[5])/3;
		
		get.OutputField.r_Frequency	:= DataBuffer[25];
		
		CASE REAL_TO_INT(DataBuffer[26]) OF
			-1 	:	get.OutputField.e_ACrotationStatus := eACRotationState.Left;
			1	:	get.OutputField.e_ACrotationStatus := eACRotationState.Right;
			0	:	get.OutputField.e_ACrotationStatus := eACRotationState.None;
		END_CASE

		//field specific data, keep separate at first. Then combine data into get struct in a later step.
		get.OutputField.ar_PowerlockCurrents[1][Phases.L1] := DataBuffer[6];
		get.OutputField.ar_PowerlockCurrents[1][Phases.L2] := DataBuffer[7];
		get.OutputField.ar_PowerlockCurrents[1][Phases.L3] := DataBuffer[8];
		get.OutputField.ar_PowerlockCurrents[1][Phases.N] := DataBuffer[9];
		
		ast_OutputPowerLockData[1].r_ActivePhasePower[phases.L1] := DataBuffer[10];
   		ast_OutputPowerLockData[1].r_ActivePhasePower[phases.L2] := DataBuffer[11];
		ast_OutputPowerLockData[1].r_ActivePhasePower[phases.L3] := DataBuffer[12];
		ast_OutputPowerLockData[1].r_ActivePhasePower[phases.AVG] := (DataBuffer[10] + DataBuffer[11] + DataBuffer[12])/3;
		                        
		ast_OutputPowerLockData[1].r_ApparentPhasePower[phases.L1] := DataBuffer[14];
   		ast_OutputPowerLockData[1].r_ApparentPhasePower[phases.L2] := DataBuffer[15];
		ast_OutputPowerLockData[1].r_ApparentPhasePower[phases.L3] := DataBuffer[16];
		ast_OutputPowerLockData[1].r_ApparentPhasePower[phases.AVG] := (DataBuffer[14] + DataBuffer[15] + DataBuffer[16])/3;
		                        
		ast_OutputPowerLockData[1].r_ReactivePhasePower[phases.L1] := DataBuffer[18];
   		ast_OutputPowerLockData[1].r_ReactivePhasePower[phases.L2] := DataBuffer[19];
		ast_OutputPowerLockData[1].r_ReactivePhasePower[phases.L3] := DataBuffer[20];
		ast_OutputPowerLockData[1].r_ReactivePhasePower[phases.AVG] := (DataBuffer[18] + DataBuffer[19] + DataBuffer[20])/3;
		    				                        
		ast_OutputPowerLockData[1].r_ActivePower := DataBuffer[13];
		ast_OutputPowerLockData[1].r_ApparentPower := DataBuffer[17];
		ast_OutputPowerLockData[1].r_ReactivePower := DataBuffer[21];

		ast_OutputPowerLockData[1].ar_PowerFactor[Phases.L1] := DataBuffer[22];
		ast_OutputPowerLockData[1].ar_PowerFactor[Phases.L2] := DataBuffer[23];
		ast_OutputPowerLockData[1].ar_PowerFactor[Phases.L3] := DataBuffer[24];
		ast_OutputPowerLockData[1].ar_PowerFactor[Phases.AVG] := (DataBuffer[22] + DataBuffer[23] + DataBuffer[24])/3;
		
		ast_OutputPowerLockData[1].r_EnergyConsumed	:=  DataBuffer[34];
		ast_OutputPowerLockData[1].r_EnergySupplied 	:=	DataBuffer[38];

		ast_OutputPowerLockData[1].ar_THD[Phases.L1] := DataBuffer[58];
		ast_OutputPowerLockData[1].ar_THD[Phases.L2] := DataBuffer[59];
		ast_OutputPowerLockData[1].ar_THD[Phases.L3] := DataBuffer[60];
			
		ui_MBRetryCount := 0;
		sfctip := TRUE;
	ELSE
		ui_MBRetryCount := ui_MBRetryCount + 1;
		
		IF ui_MBRetryCount > 1 THEN
			get.events.b_MBCommWarning := TRUE;
		END_IF	
		
		//if comm fails 5 times in a row. try next input
		IF ui_MBRetryCount > 4 THEN
			get.Events.b_MBCommError := TRUE;
			sfctip := TRUE;
		END_IF
	END_IF
END_IF
END_ACTION

ACTION aReadOutputField2:

MBRead(
sIPAddr := PowerMeterConfig.IP_JANITZA,
nTCPPort := PowerMeterConfig.MBPort_Janitza,
nUnitID := 1,//16#FF,
nMBAddr := 19200,
nQuantity := 50*2,
cbLength := SIZEOF(DataBuffer),
pDestAddr := ADR(DataBuffer),
bExecute := NOT (b_busy OR TransmissionDone.Q),	//	<- werkt dit niet gewoon?
bBusy => b_busy,
bError => b_CommError,
nErrId => udi_errid,
cbRead => udi_cbread,
tTimeout := T#25MS
);

TransmissionDone(clk := b_busy);

IF TransmissionDone.q THEN
	IF NOT b_CommError THEN	
		
		FOR UI_Iterator := 0 TO 50 BY 1 DO
			DataBuffer[UI_Iterator] := ChangeRealEndianess(DataBuffer[UI_Iterator]);
		END_FOR 	
	
		get.OutputField.ar_PowerlockCurrents[2][Phases.L1] := DataBuffer[0];
		get.OutputField.ar_PowerlockCurrents[2][Phases.L2] := DataBuffer[1];
		get.OutputField.ar_PowerlockCurrents[2][Phases.L3] := DataBuffer[2];
		get.OutputField.ar_PowerlockCurrents[2][Phases.N] := DataBuffer[3];

		ast_OutputPowerLockData[2].r_ActivePhasePower[phases.L1] := DataBuffer[4];
   		ast_OutputPowerLockData[2].r_ActivePhasePower[phases.L2] := DataBuffer[5];
		ast_OutputPowerLockData[2].r_ActivePhasePower[phases.L3] := DataBuffer[6];
		ast_OutputPowerLockData[2].r_ActivePhasePower[phases.AVG] := (DataBuffer[4] + DataBuffer[5] + DataBuffer[6])/3;
		
		ast_OutputPowerLockData[2].r_ApparentPhasePower[phases.L1] := DataBuffer[8];
   		ast_OutputPowerLockData[2].r_ApparentPhasePower[phases.L2] := DataBuffer[9];
		ast_OutputPowerLockData[2].r_ApparentPhasePower[phases.L3] := DataBuffer[10];
		ast_OutputPowerLockData[2].r_ApparentPhasePower[phases.AVG] := (DataBuffer[8] + DataBuffer[9] + DataBuffer[10])/3;
		
		ast_OutputPowerLockData[2].r_ReactivePhasePower[phases.L1] := DataBuffer[12];
   		ast_OutputPowerLockData[2].r_ReactivePhasePower[phases.L2] := DataBuffer[13];
		ast_OutputPowerLockData[2].r_ReactivePhasePower[phases.L3] := DataBuffer[14];
		ast_OutputPowerLockData[2].r_ReactivePhasePower[phases.AVG] := (DataBuffer[12] + DataBuffer[13] + DataBuffer[14])/3;
		    				                        
		ast_OutputPowerLockData[2].r_ActivePower := DataBuffer[7];
		ast_OutputPowerLockData[2].r_ApparentPower := DataBuffer[11];
		ast_OutputPowerLockData[2].r_ReactivePower := DataBuffer[15];
                                
		ast_OutputPowerLockData[2].ar_PowerFactor[Phases.L1] := DataBuffer[16];
		ast_OutputPowerLockData[2].ar_PowerFactor[Phases.L2] := DataBuffer[17];
		ast_OutputPowerLockData[2].ar_PowerFactor[Phases.L3] := DataBuffer[18];
		ast_OutputPowerLockData[2].ar_PowerFactor[Phases.AVG] := (DataBuffer[16] + DataBuffer[17] + DataBuffer[18])/3;
		                        
		ast_OutputPowerLockData[2].r_EnergyConsumed	:=  DataBuffer[26];
		ast_OutputPowerLockData[2].r_EnergySupplied 	:=	DataBuffer[30];
				                
		ast_OutputPowerLockData[2].ar_THD[Phases.L1] := DataBuffer[47];
		ast_OutputPowerLockData[2].ar_THD[Phases.L2] := DataBuffer[48];
		ast_OutputPowerLockData[2].ar_THD[Phases.L3] := DataBuffer[49];
			
		ui_MBRetryCount := 0;
		sfctip := TRUE;
	ELSE
		ui_MBRetryCount := ui_MBRetryCount + 1;
		
		IF ui_MBRetryCount > 1 THEN
			get.events.b_MBCommWarning := TRUE;
		END_IF	
		
		//if comm fails 5 times in a row. try next input
		IF ui_MBRetryCount > 4 THEN
			get.Events.b_MBCommError := TRUE;
			sfctip := TRUE;
		END_IF
	END_IF
END_IF
END_ACTION

ACTION aReadOutputField3:

IF NOT PowerMeterConfig.b_ThirdOutputFieldAvailable THEN
	//skip this step if third field isn't in use
	SFCTip := TRUE;
ELSE
	MBRead(
	sIPAddr := PowerMeterConfig.IP_JANITZA,
	nTCPPort := PowerMeterConfig.MBPort_Janitza,
	nUnitID := 1,//16#FF;
	nMBAddr := 19400,
	nQuantity := 50*2,
	cbLength := SIZEOF(SecondDataBuffer),
	pDestAddr := ADR(SecondDataBuffer),
	bExecute := NOT (b_busy OR TransmissionDone.Q),	//	<- werkt dit niet gewoon?
	bBusy => b_busy,
	bError => b_CommError,
	nErrId => udi_errid,
	cbRead => udi_cbread,
	tTimeout := T#25MS
	);
	
	TransmissionDone(clk := b_busy);
	
	IF TransmissionDone.q THEN
		IF NOT b_CommError  THEN	
			
			FOR UI_Iterator := 0 TO 50 BY 1 DO
				DataBuffer[UI_Iterator] := ChangeRealEndianess(SecondDataBuffer[UI_Iterator]);
			END_FOR 
			//field specific data, keep separate at first. Then combine data into get struct in a later step.
			get.OutputField.ar_PowerlockCurrents[3][Phases.L1] := DataBuffer[0];
			get.OutputField.ar_PowerlockCurrents[3][Phases.L2] := DataBuffer[1];
			get.OutputField.ar_PowerlockCurrents[3][Phases.L3] := DataBuffer[2];
			get.OutputField.ar_PowerlockCurrents[3][Phases.N] := DataBuffer[3];

			ast_OutputPowerLockData[3].r_ActivePhasePower[phases.L1] := DataBuffer[4];
 	  		ast_OutputPowerLockData[3].r_ActivePhasePower[phases.L2] := DataBuffer[5];
			ast_OutputPowerLockData[3].r_ActivePhasePower[phases.L3] := DataBuffer[6];
			ast_OutputPowerLockData[3].r_ActivePhasePower[phases.AVG] := (DataBuffer[4] + DataBuffer[5] + DataBuffer[6])/3;
		                            
			ast_OutputPowerLockData[3].r_ApparentPhasePower[phases.L1] := DataBuffer[8];
	   		ast_OutputPowerLockData[3].r_ApparentPhasePower[phases.L2] := DataBuffer[9];
			ast_OutputPowerLockData[3].r_ApparentPhasePower[phases.L3] := DataBuffer[10];
			ast_OutputPowerLockData[3].r_ApparentPhasePower[phases.AVG] := (DataBuffer[8] + DataBuffer[9] + DataBuffer[10])/3;
		                            
			ast_OutputPowerLockData[3].r_ReactivePhasePower[phases.L1] := DataBuffer[12];
 	 		ast_OutputPowerLockData[3].r_ReactivePhasePower[phases.L2] := DataBuffer[13];
			ast_OutputPowerLockData[3].r_ReactivePhasePower[phases.L3] := DataBuffer[14];
			ast_OutputPowerLockData[3].r_ReactivePhasePower[phases.AVG] := (DataBuffer[12] + DataBuffer[13] + DataBuffer[14])/3;
		    				                        
			ast_OutputPowerLockData[3].r_ActivePower := DataBuffer[7];
			ast_OutputPowerLockData[3].r_ApparentPower := DataBuffer[11];
			ast_OutputPowerLockData[3].r_ReactivePower := DataBuffer[15];
									
			ast_OutputPowerLockData[3].ar_PowerFactor[Phases.L1] := DataBuffer[16];
			ast_OutputPowerLockData[3].ar_PowerFactor[Phases.L2] := DataBuffer[17];
			ast_OutputPowerLockData[3].ar_PowerFactor[Phases.L3] := DataBuffer[18];
			ast_OutputPowerLockData[3].ar_PowerFactor[Phases.AVG] := (DataBuffer[16] + DataBuffer[17] + DataBuffer[18])/3;
									
			ast_OutputPowerLockData[3].r_EnergyConsumed	:=  DataBuffer[26];
			ast_OutputPowerLockData[3].r_EnergySupplied 	:=	DataBuffer[30];
									
			ast_OutputPowerLockData[3].ar_THD[Phases.L1] := DataBuffer[47];
			ast_OutputPowerLockData[3].ar_THD[Phases.L2] := DataBuffer[48];
			ast_OutputPowerLockData[3].ar_THD[Phases.L3] := DataBuffer[49];
				
			ui_MBRetryCount := 0;
			sfctip := TRUE;
		ELSE
			ui_MBRetryCount := ui_MBRetryCount + 1;

			IF ui_MBRetryCount > 1 THEN
				get.events.b_MBCommWarning := TRUE;
			END_IF	
			
			//if comm fails 5 times in a row. try next input
			IF ui_MBRetryCount > 4 THEN
				get.Events.b_MBCommError := TRUE;
				sfctip := TRUE;
			END_IF
		END_IF
	END_IF
END_IF
END_ACTION

METHOD ChangeRealEndianess : REAL
VAR_INPUT
	InputReal	:	REAL;
END_VAR

VAR
	TestWord	:	WORD;
	TestByte	: ARRAY[0..3] OF BYTE;
END_VAR

MEMCPY(ADR(ChangeRealEndianess)+2, 	ADR(InputReal), 	2);
MEMCPY(ADR(ChangeRealEndianess), 	ADR(InputReal)+2, 	2);

memcpy(ADR(TestWord), ADR(InputReal), 2);
IF ((TestWord AND 2#0111111110000000) = 2#0111111110000000) THEN
	ChangeRealEndianess := 0;
END_IF
END_METHOD

ACTION ReadDataSFC:
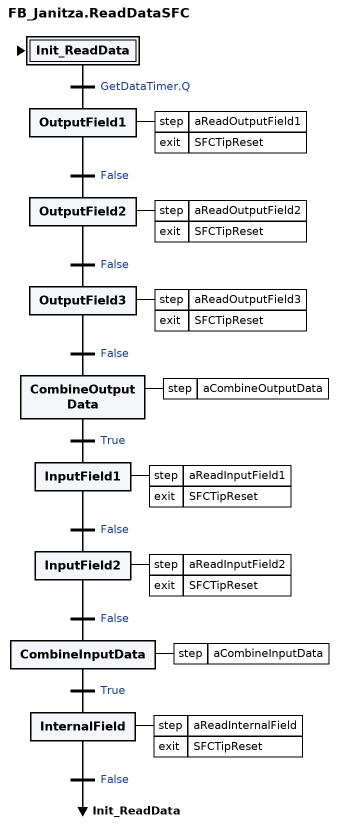
INITIAL_STEP Init_ReadData:
END_STEP
TRANSITION FROM Init_ReadData TO OutputField1
    := GetDataTimer.Q;
END_TRANSITION
STEP OutputField1:
    aReadOutputField1(N);  // step action
    SFCTipReset(P0);  // exit action
END_STEP
TRANSITION FROM OutputField1 TO OutputField2
    := False;
END_TRANSITION
STEP OutputField2:
    aReadOutputField2(N);  // step action
    SFCTipReset(P0);  // exit action
END_STEP
TRANSITION FROM OutputField2 TO OutputField3
    := False;
END_TRANSITION
STEP OutputField3:
    aReadOutputField3(N);  // step action
    SFCTipReset(P0);  // exit action
END_STEP
TRANSITION FROM OutputField3 TO CombineOutputData
    := False;
END_TRANSITION
STEP CombineOutputData:
    aCombineOutputData(N);  // step action
END_STEP
TRANSITION FROM CombineOutputData TO InputField1
    := True;
END_TRANSITION
STEP InputField1:
    aReadInputField1(N);  // step action
    SFCTipReset(P0);  // exit action
END_STEP
TRANSITION FROM InputField1 TO InputField2
    := False;
END_TRANSITION
STEP InputField2:
    aReadInputField2(N);  // step action
    SFCTipReset(P0);  // exit action
END_STEP
TRANSITION FROM InputField2 TO CombineInputData
    := False;
END_TRANSITION
STEP CombineInputData:
    aCombineInputData(N);  // step action
END_STEP
TRANSITION FROM CombineInputData TO InternalField
    := True;
END_TRANSITION
STEP InternalField:
    aReadInternalField(N);  // step action
    SFCTipReset(P0);  // exit action
END_STEP
TRANSITION FROM InternalField TO Init_ReadData
    := False;
END_TRANSITION
END_ACTION

ACTION SFCTipReset:
SFCTip := FALSE;
END_ACTION

END_FUNCTION_BLOCK

// ---- POUs/Objects/PowerQualityMonitor/FB_PowerQualityMonitoring.TcPOU
FUNCTION_BLOCK FB_PowerQualityMonitoring
VAR_OUTPUT
	get						: ST_PowerMonitor_get;
END_VAR

VAR_INPUT
	b_Enable		: 	BOOL;
	PowerStackGet	:	st_Powerstack_Get;	// change into reference?
	b_TNModeActive	:	BOOL;
END_VAR

VAR
	Janitza: FB_Janitza;
	El3443: FB_EL3443_0010;
END_VAR

VAR CONSTANT
	w_ID : WORD := 1;//:= eObject_ID.PowerMonitor;
END_VAR

(*
Update rate is 200 ms max.
So call IO method only every 200ms.
More calls only increase cpu and network load.
*)

//get data from janitza powermeter
Janitza(get:=get, ReadData:=b_Enable, b_TNmodeEnable := b_TNModeActive);
EL3443(get:=get, b_Enable:=b_Enable);

//Voltage dependent values of Internal supply are copied from outputfield, but are only valid if netcontactor is closed.
IF (PowerStackGet.e_NetContactorStatus = eNetcontactorState.LeftClosed) OR 
	(PowerStackGet.e_NetContactorStatus = eNetcontactorState.RightClosed) THEN
	get.InternalSupply.e_ACrotationStatus := get.OutputField.e_ACrotationStatus;
	get.InternalSupply.r_LineVoltage := get.OutputField.r_LineVoltage;
	get.InternalSupply.r_PhaseVoltage := get.OutputField.r_PhaseVoltage;
	get.InternalSupply.r_Frequency := get.OutputField.r_Frequency;
ELSE
	get.InternalSupply.e_ACrotationStatus 	:= 	eACRotationSTate.None;
	
	get.InternalSupply.r_LineVoltage[phases.L1] 		:= 	0;
	get.InternalSupply.r_LineVoltage[phases.L2] 		:= 	0;
	get.InternalSupply.r_LineVoltage[phases.L3] 		:= 	0;
	get.InternalSupply.r_LineVoltage[phases.AVG] 		:= 	0;
	
	get.InternalSupply.r_PhaseVoltage[phases.L1] 		:= 	0;
	get.InternalSupply.r_PhaseVoltage[phases.L2] 		:= 	0;
	get.InternalSupply.r_PhaseVoltage[phases.L3] 		:= 	0;
	get.InternalSupply.r_PhaseVoltage[phases.AVG] 		:= 	0;
	
	get.InternalSupply.r_Frequency						:= 	0;
END_IF



//Fill BESS data with PowerStackData
//Not all data is filled in here, determine which are desired and possible.

//phase currents not available at this time, only the average is set
get.BESS.r_Current[Phases.AVG] := PowerStackGet.r_AcCurrent;

//phase Powers not available at this time, only the average is set
Get.BESS.r_ApparentPower	:=	PowerStackGet.r_ApparentPower;
Get.BESS.r_ReactivePower	:=	PowerStackGet.r_ReactivePower;
Get.BESS.r_ActivePower		:=	PowerStackGet.r_ActivePower;
	
Get.BESS.r_Frequency		:=  PowerStackGet.r_ACSupplyFrequency;

//phase Powerfactors not available at this time, only the average is set									
Get.BESS.r_PowerFactor[Phases.AVG]		:=	PowerStackGet.r_CosPhi;

METHOD PUBLIC EMstop : BOOL
//returns true when ready/stopped
END_METHOD

METHOD GetDiagnostics
VAR_IN_OUT
	AddError		: ARRAY [*] OF FB_AddErrorST;
	a_ActiveEvents	: ARRAY [*] OF ST_ErrorStruct;
	w_Index			: WORD;
END_VAR

VAR_OUTPUT
	b_errorActive	: BOOL;
	b_warningActive	: BOOL;
END_VAR

VAR
	by_errCt	: BYTE;
	by_warnCt	: BYTE;
END_VAR
//JANITZA
(*Comm Warning*)		AddError[w_Index](
		in_b_ErrorTrig			:= get.events.b_MBCommWarning,
		out_ST_Error			:= a_ActiveEvents[w_Index],
		w_ID					:= 1 + w_ID,
		s_Message				:= 'PowerQualityMonitor communication warning',
		e_sev					:= eseverity.warning
	);
	IF AddError[w_Index].b_out THEN by_warnCt := by_warnCt + 1; END_IF;
	w_Index := w_Index +1;
	
(*Comm timeout*)		AddError[w_Index](
		in_b_ErrorTrig			:= get.events.b_MBTimeoutWarning,
		out_ST_Error			:= a_ActiveEvents[w_Index],
		w_ID					:= 2 + w_ID,
		s_Message				:= 'PowerQualityMonitor communication timeout',
		e_sev					:= eseverity.Warning
	);
	IF AddError[w_Index].b_out THEN by_warnCt := by_warnCt + 1; END_IF;
	w_Index := w_Index +1;
	
(*Comm fault*)		AddError[w_Index](
		in_b_ErrorTrig			:= get.events.b_MBCommError,
		out_ST_Error			:= a_ActiveEvents[w_Index],
		w_ID					:= 3 + w_ID,
		in_t_triggerTime		:= T#10S,
		s_Message				:= 'PowerQualityMonitor communication fault',
		e_sev					:= eseverity.Normalshutdown
	);
	IF AddError[w_Index].b_out THEN by_errCt := by_errCt + 1; END_IF;
	w_Index := w_Index +1;
	
//EL3443
(*Comm Warning*)		AddError[w_Index](
		in_b_ErrorTrig			:= get.events.b_EL3443Warning,
		out_ST_Error			:= a_ActiveEvents[w_Index],
		w_ID					:= 4 + w_ID,
		s_Message				:= 'EL3443 powermonitor warning',
		e_sev					:= eseverity.Warning
	);
	IF AddError[w_Index].b_out THEN by_warnCt := by_warnCt + 1; END_IF;
	w_Index := w_Index +1;
	
(*Comm Fault*)		AddError[w_Index](
		in_b_ErrorTrig			:= get.events.b_EL3443Error,
		out_ST_Error			:= a_ActiveEvents[w_Index],
		w_ID					:= 5 + w_ID,
		s_Message				:= 'EL3443 powermonitor fault',
		e_sev					:= eseverity.NormalShutdown
	);
	IF AddError[w_Index].b_out THEN by_errCt := by_errCt + 1; END_IF;
	w_Index := w_Index +1;

b_errorActive := by_errCt <>0;
b_warningActive := by_warnCt <>0;
END_METHOD

METHOD Public Reset : BOOL
//clear data struct
//reinitialize janitza + el3443
//clear all errors?

//returns true when ready
END_METHOD

END_FUNCTION_BLOCK

// ---- POUs/Objects/ProtectionSystems/FireDetection/FB_FireDetection.TcPOU
FUNCTION_BLOCK FB_FireDetection
VAR_OUTPUT
	Get	:	ST_FireDetectionGet;
END_VAR

VAR_INPUT
	TestSounder		AT %I* : BOOL;
	//Set	:	ST_FireDetectionSet;
END_VAR

VAR
	SmokeDetIO				:	ST_SmokeDetIO;
	CODetMeasValues			:	ARRAY[1..2] OF REAL;
	b_SounderOn				:	BOOL	:= FALSE;
	b_SilenceSounder	 	:	BOOL;
	b_ResetSystem		 	:	BOOL;
END_VAR

VAR
	//w_ID							: WORD := eObject_ID.FireDetection;
	IO								: FB_FireDetection_IO;
	//Diagnostics						: FB_FireDetection_Diagnostics;
END_VAR

(*
IO(
	r_CODet1_value => get.CODetectorValues[1],
	r_CODet2_value => get.CODetectorValues[2],
	b_SmokeDetectorSignal_OK => ,
	b_SmokeDetectorPower_OK
	
	);
	
 SmokeDetIO:=SmokeDetIO, b_SounderOn:=b_SounderOn);

CheckSmokeDetectors();
CheckCODetectors();
SounderBeacon();
Reset();
Diagnostics();
//ResetDetectors(b_ResetAlarms);

//CAll diagnostics
(*diagnostics(
	w_ID := w_ID,
	w_ErrorIndex := w_ErrorIndex, 
	AddError:=AddError,
	w_ErrorControlWord := w_ErrorControLWord	
);
*)
//diagnostic toevoegen: warning if reset input remains high after reset timeout
*)

METHOD PRIVATE CheckCODetectors : BOOL


VAR_inst
	//short term average filter for CO detector 1 (100ms)
	CO_DET1_Avg: FB_CTRL_MOVING_AVERAGE := (fTaskCycleTime := 1.0, fCtrlCycleTime := 1.0);
	CO_DET1_AVG_PARAMS	:	ST_CTRL_MOVING_AVERAGE_PARAMS := (tCtrlCycleTime := TIME#1MS, tTaskCycleTime := TIME#1MS, nSamplesToFilter := 10, pWorkArray_ADR := ADR(CO_DET1_Values[1]), nWorkArray_SIZEOF := SIZEOF(CO_DET1_Values));

	
	//short term average filter for CO detector 2 (100ms)
	CO_DET2_Avg: FB_CTRL_MOVING_AVERAGE := (fTaskCycleTime := 1.0, fCtrlCycleTime := 1.0);
	CO_DET2_AVG_PARAMS	:	ST_CTRL_MOVING_AVERAGE_PARAMS := (tCtrlCycleTime := TIME#1MS, tTaskCycleTime := TIME#1MS, nSamplesToFilter := 10, pWorkArray_ADR := ADR(CO_DET2_Values[1]), nWorkArray_SIZEOF := SIZEOF(CO_DET2_Values));
	
	
	Warning1Timer	:	TON := (PT := TIME#1H);
	Warning2Timer	:	TON := (PT := TIME#15m);
END_VAR

VAR

END_VAR

//actual sensor value already filled in in IO code. Only generate status data here.
//alarm status can not be cleared in this method. only via fb_firedetection.reset method.
//alarm status is te highest status, if true, no work to do here.

//if both sensors are working
IF (get.CODetectorValues[1] > -1) AND (get.CODetectors.CODetectorValues[2] > -1) THEN
	IF get.CODetectors.CODetectorState = eCOAlarmStatus.Error THEN
		get.CODetectors.CODetectorState := eCOAlarmStatus.Normal;
	END_IF
	
	get.CODetectors.CODetectorValues[1] := CODetMeasValues[1];
	get.CODetectors.CODetectorValues[2] := CODetMeasValues[2];
	get.CODetectors.CODetectorValues[0] := (CODetMeasValues[1]/2) + (CODetMeasValues[2]/2);
	
ELSE
	//at least 1 detector is faulty, so go to error state
	IF get.CODetectors.CODetectorState = eCOAlarmStatus.Normal THEN
		get.CODetectors.CODetectorState := eCOAlarmStatus.Error;
	END_IF
	
	//if only sensor 1 working
	IF (get.CODetectors.CODetectorValues[1] > -1) AND (get.CODetectors.CODetectorValues[2] = -1) THEN
		get.CODetectors.CODetectorValues[1] := CODetMeasValues[1];
		get.CODetectors.CODetectorValues[2] := -1;
		get.CODetectors.CODetectorValues[0] := (CODetMeasValues[1]);

	//if only sensor 2 working
	ELSIF (get.CODetectors.CODetectorValues[2] > -1) AND (get.CODetectors.CODetectorValues[1] = -1) THEN

		get.CODetectors.CODetectorValues[1] := -1;
		get.CODetectors.CODetectorValues[2] := CODetMeasValues[2];
		get.CODetectors.CODetectorValues[0] := CODetMeasValues[2];
	//nothing working
	ELSE
		get.CODetectors.CODetectorValues[0] := -1;
		get.CODetectors.CODetectorValues[1] := -1;
		get.CODetectors.CODetectorValues[2] := -1;
	END_IF
END_IF

//thermal runaway can be triggered by 1 sensor as this can be localized issue which may take time to spread.
IF (get.CODetectors.CODetectorValues[1] > 120) OR (get.CODetectors.CODetectorValues[2] > 120) THEN
	get.Events.b_CODetAlarm := TRUE;
END_IF

//Warning levels are no longer triggered based on an average
//pgs-37 requires separate triggers per sensor.
Warning1Timer(IN := (get.CODetectors.CODetectorValues[1] > 10) OR (get.CODetectors.CODetectorValues[2] > 10));
get.Events.b_CODetWarning2 := Warning2Timer.Q;

Warning2Timer(IN := (get.CODetectors.CODetectorValues[1] > 20) OR (get.CODetectors.CODetectorValues[2] > 20));
get.Events.b_CODetWarning1 := Warning1Timer.Q;
END_METHOD

METHOD PRIVATE CheckSmokeDetectors

VAR_INST
	AlarmResetTimer: TP := (PT := TIME#500MS);
	SmokeAlarmTimer: TON := (PT := TIME#500ms);
	AlarmResetTrigger: F_TRIG;
	SmokeAlarmPowerLost: TON := (PT := TIME#50MS);
END_VAR


//input delay for alarm inputs
SmokeAlarmTimer(IN := (NOT SmokeDetIO.SmokeDetectorSignal_OK) AND (NOT AlarmResetTrigger.Q));
SmokeAlarmPowerLost(IN := (NOT SmokeDetIO.SmokeDetectorPower_OK) AND  (NOT AlarmResetTrigger.Q));

IF get.SmokeDetectors.SmokeDetectorState = efireAlarmstatus.Normal THEN
	IF SmokeAlarmPowerLost.Q THEN	//Alarm power failure means alarm cannot be trusted. So first check power
		get.SmokeDetectors.SmokeDetectorState := efireAlarmstatus.Error;
	ELSIF SmokeAlarmTimer.Q THEN	//if alarm signals for >500ms --> raise the alarm.
		get.SmokeDetectors.SmokeDetectorState := efireAlarmstatus.Alarm;	//alarm is only resettable manually via resetDetectors
	END_IF
ELSIF get.SmokeDetectors.SmokeDetectorState = efireAlarmstatus.Error THEN	//if power failed, no alarm checking anymore as this will give false alarms
	IF NOT SmokeAlarmPowerLost.Q THEN	//Alarm state may return to operational if power comes back
		get.SmokeDetectors.SmokeDetectorState := efireAlarmstatus.Normal;
	END_IF
END_IF	//In alarm state, no power checking is performed anymore. Even if the detectors lose power now, the alarm state has priority.
END_METHOD

METHOD Diagnostics : BOOL
VAR_INPUT
END_VAR

get.Events.SmokeDetAlarm 	:= (get.SmokeDetectors.SmokeDetectorState = eFireAlarmStatus.Alarm);
get.Events.SmokeDetFault 	:= (get.SmokeDetectors.SmokeDetectorState = eFireAlarmStatus.Error);
get.Events.CODetAlarm 		:= (get.CODetectors.CODetectorState = eCOAlarmStatus.Alarm);
get.Events.CODetFault 		:= (get.CODetectors.CODetectorState = eCOAlarmStatus.Error);
get.Events.CODetWarning		:= (get.CODetectors.CODetectorState = eCOAlarmStatus.WarningLevel1)OR(get.CODetectors.CODetectorState = eCOAlarmStatus.WarningLevel2);

get.Events.AlarmMuted 		:= (get.Events.SmokeDetAlarm OR get.Events.CODetAlarm) And not SounderOn;
END_METHOD

METHOD PUBLIC EMstop : BOOL
VAR_INPUT
END_VAR
//do anything?
//return true when ready
END_METHOD

METHOD PUBLIC Reset : BOOL
VAR_INPUT
//	ResetActive : BOOL := FALSE;
END_VAR

VAR_INST
	SmokeDetPowerDownTimer : TP := (PT := TIME#250MS);
	PowerUpTrigger	:	f_trig;
	ResetTrigger	:	r_trig;
END_VAR
//reset detectors
//return true when ready

SounderOn;

Reset := FALSE; 
SmokeDetPowerDownTimer(IN := ResetSystem);
SmokeDetIO.SmokeDetectorShutdown := SmokeDetPowerDownTimer.Q;

PowerUpTrigger(CLK := SmokeDetPowerDownTimer.Q);
IF PowerUpTrigger.Q THEN
	get.SmokeDetectors.SmokeDetectorState := eFireAlarmStatus.Normal;
	Reset := TRUE; 
END_IF

ResetTrigger(CLK := ResetSystem);
IF ResetTrigger.Q THEN
	get.CODetectors.CODetectorState := eCOAlarmStatus.Normal;
END_IF

SilenceSounder := ResetTrigger.Q;
END_METHOD

METHOD SounderBeacon : BOOL

VAR_INST
	Old_COAlarmState	:	BOOL := FALSE;
	Old_SmokeAlarmState	:	BOOL := FALSE;
	SilenceTrigger : R_Trig;
	TestTrigger : R_Trig;
END_VAR

//Only enable sounder at the start of the alarm. Use old_state to determine this.
//This allows for alarm muting and retriggering. 

IF NOT old_COAlarmState THEN
	IF get.CODetectors.CODetectorState = eCOAlarmStatus.Alarm THEN
		SounderOn := TRUE;
		old_COAlarmState := TRUE;
	END_IF
ELSE
	IF get.CODetectors.CODetectorState = eCOAlarmStatus.Normal THEN
		old_COAlarmState := FALSE;
	END_IF			
END_IF

IF NOT old_SmokeAlarmState THEN
	IF get.SmokeDetectors.SmokeDetectorState = eFireAlarmStatus.Alarm THEN
		SounderOn := TRUE;
		old_SmokeAlarmState := TRUE;
	END_IF
ELSE
	IF get.SmokeDetectors.SmokeDetectorState = eFireAlarmStatus.Normal THEN
		old_SmokeAlarmState := FALSE;
	END_IF		
END_IF

//use rtrig to prevent permanent muting.
SilenceTrigger(clk:= SilenceSounder);
IF SilenceTrigger.Q THEN
	SounderOn := FALSE;
END_IF

//use rtrig to prevent permanent sounding. resilence with muting.
TestTrigger(clk:= TestSounder);
IF TestTrigger.Q THEN
	SounderOn := TRUE;
END_IF
END_METHOD

END_FUNCTION_BLOCK

// ---- POUs/Objects/ProtectionSystems/FireDetection/FB_FireDetection_IO.TcPOU
FUNCTION_BLOCK FB_FireDetection_IO

VAR_OUTPUT
	r_CODet1_value				: REAL;
	r_CODet2_value				: REAL;
	b_SmokeDetectorSignal_OK 	: BOOL;
	b_SmokeDetectorPower_OK 	: BOOL;
END_VAR

VAR
	SmokeDetPwr			AT %Q* 	: BOOL;	
	SmokeDetSts			AT %I* 	: ARRAY[1..2] OF BOOL;
	CO_read				AT %I*	: ARRAY [1..2] OF ST_COInputData;
	SounderOut			AT %Q* 	: BOOL;	
END_VAR

VAR_INPUT
	b_DisableSmokeDetectors		: BOOL;
	b_SounderOn					: BOOL;
END_VAR


CO_detector_IO();
Smoke_detector_IO();
sounder_IO();

METHOD CO_detector_IO : BOOL
VAR
	ScaleCOValue: FB_CTRL_SCALE;
	COScaleParams: ST_CTRL_SCALE_PARAMS := (tTaskCycleTime := TIME#1ms, fInMin := 0, fInMax := 4095, fOutMax := 200.0);
END_VAR
IF CO_read[1].b_InputOverrange OR CO_read[1].b_InputUnderrange THEN
	r_CODet1_value := -1;
ELSE
	//ScaleCOValue(fIn := CO_read[1].Value, stParams:= COScaleParams, fOut=>Get.CODetectors.CODetectorValue[1]);
	r_CODet1_value := CO_read[1].w_Value/20.475;
END_IF

IF CO_read[2].b_InputOverrange OR CO_read[2].b_InputUnderrange THEN
	r_CODet2_value := -1;
ELSE
	r_CODet2_value := CO_read[2].w_Value/20.475;
	//ScaleCOValue(fIn := CO_read[2].Value, stParams:= COScaleParams, fOut=>Get.CODetectors.CODetectorValue[2]);
END_IF
END_METHOD

METHOD Smoke_Detector_IO : BOOL
VAR_INPUT
END_VAR
b_SmokeDetectorSignal_OK 	:= SmokeDetSts[1];
b_SmokeDetectorPower_OK 	:= SmokeDetSts[2];

SmokeDetPwr := b_DisableSmokeDetectors;
END_METHOD

METHOD Sounder_IO : BOOL
SounderOut := SounderOn;
END_METHOD

END_FUNCTION_BLOCK

// ---- POUs/old/old.TcPOU
FUNCTION_BLOCK old
VAR_INPUT
END_VAR
VAR_OUTPUT
END_VAR
VAR
END_VAR

ACTION BMSInit:
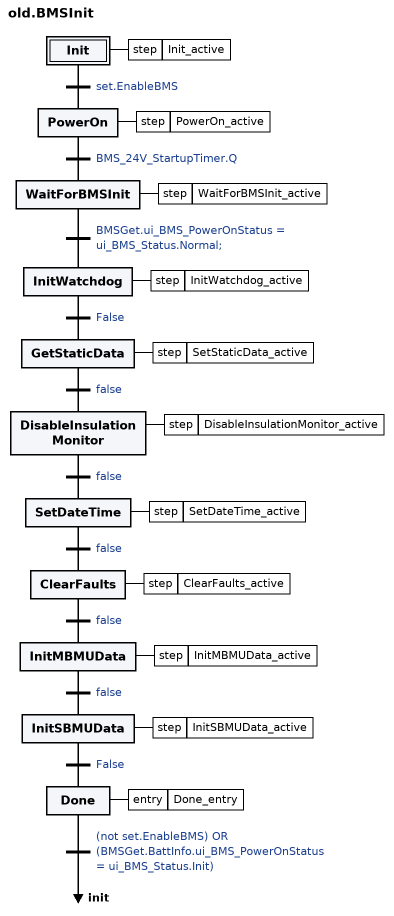
INITIAL_STEP Init:
    Init_active(N);  // step action
END_STEP
TRANSITION FROM Init TO PowerOn
    := set.EnableBMS;
END_TRANSITION
STEP PowerOn:
    PowerOn_active(N);  // step action
END_STEP
TRANSITION FROM PowerOn TO WaitForBMSInit
    := BMS_24V_StartupTimer.Q;
END_TRANSITION
STEP WaitForBMSInit:
    WaitForBMSInit_active(N);  // step action
END_STEP
TRANSITION FROM WaitForBMSInit TO InitWatchdog
    := BMSGet.ui_BMS_PowerOnStatus = ui_BMS_Status.Normal;
END_TRANSITION
STEP InitWatchdog:
    InitWatchdog_active(N);  // step action
END_STEP
TRANSITION FROM InitWatchdog TO GetStaticData
    := False;
END_TRANSITION
STEP GetStaticData:
    SetStaticData_active(N);  // step action
END_STEP
TRANSITION FROM GetStaticData TO DisableInsulationMonitor
    := false;
END_TRANSITION
STEP DisableInsulationMonitor:
    DisableInsulationMonitor_active(N);  // step action
END_STEP
TRANSITION FROM DisableInsulationMonitor TO SetDateTime
    := false;
END_TRANSITION
STEP SetDateTime:
    SetDateTime_active(N);  // step action
END_STEP
TRANSITION FROM SetDateTime TO ClearFaults
    := false;
END_TRANSITION
STEP ClearFaults:
    ClearFaults_active(N);  // step action
END_STEP
TRANSITION FROM ClearFaults TO InitMBMUData
    := false;
END_TRANSITION
STEP InitMBMUData:
    InitMBMUData_active(N);  // step action
END_STEP
TRANSITION FROM InitMBMUData TO InitSBMUData
    := false;
END_TRANSITION
STEP InitSBMUData:
    InitSBMUData_active(N);  // step action
END_STEP
TRANSITION FROM InitSBMUData TO Done
    := False;
END_TRANSITION
STEP Done:
    Done_entry(P1);  // entry action
END_STEP
TRANSITION FROM Done TO init
    := (not set.EnableBMS) OR (BMSGet.BattInfo.ui_BMS_PowerOnStatus = ui_BMS_Status.Init);
END_TRANSITION
END_ACTION

END_FUNCTION_BLOCK

// ---- POUs/POU.TcPOU
FUNCTION_BLOCK POU
VAR_INPUT
END_VAR
VAR_OUTPUT
END_VAR
VAR
END_VAR

//Nieuwe POU .. oke dan niet.

//Weer een toevoeging

//En nog meer features

END_FUNCTION_BLOCK

// ---- POUs/ProfinetHandling/InitSIEMENSInput.TcPOU
PROGRAM InitSIEMENSInput
VAR
	fbActPowerRQ: fbDwordToReal;
	fbReactPowerRQ: fbDwordToReal;
	fbGenActPower: fbDwordToReal;
	fbGenReactPower: fbDwordToReal;
	fbGenFreq: fbWordToReal;
	fbGenLineVoltage: fbWordToReal;
	fbMinSOCCustomer: fbWordToReal;
	fbMaxSOCCustomer: fbWordToReal;
	fbInvCurrentRampRate: fbDWordToReal;
	fbFreqDroop: fbWordToReal;
	fbVoltageDroop: fbWordToReal;
	fbInvNomVolt: fbWordToReal;
	fbInvNomFreq: fbWordToReal;
	fbCurrentLimMax: fbWordToReal;
	fbCurrentLimMin: fbWordToReal;
	fbGVoltageA		: fbWordToReal;
	fbGVoltageB		: fbWordToReal;
	fbGVoltageC		: fbWordToReal;
	fbGVoltageAB	: fbWordToReal;
	fbGVoltageBC	: fbWordToReal;
	fbGVoltageCA	: fbWordToReal;
	fbGCurrentL1	: fbWordToReal;
	fbGCurrentL2	: fbWordToReal;
	fbGCurrentL3	: fbWordToReal;
END_VAR

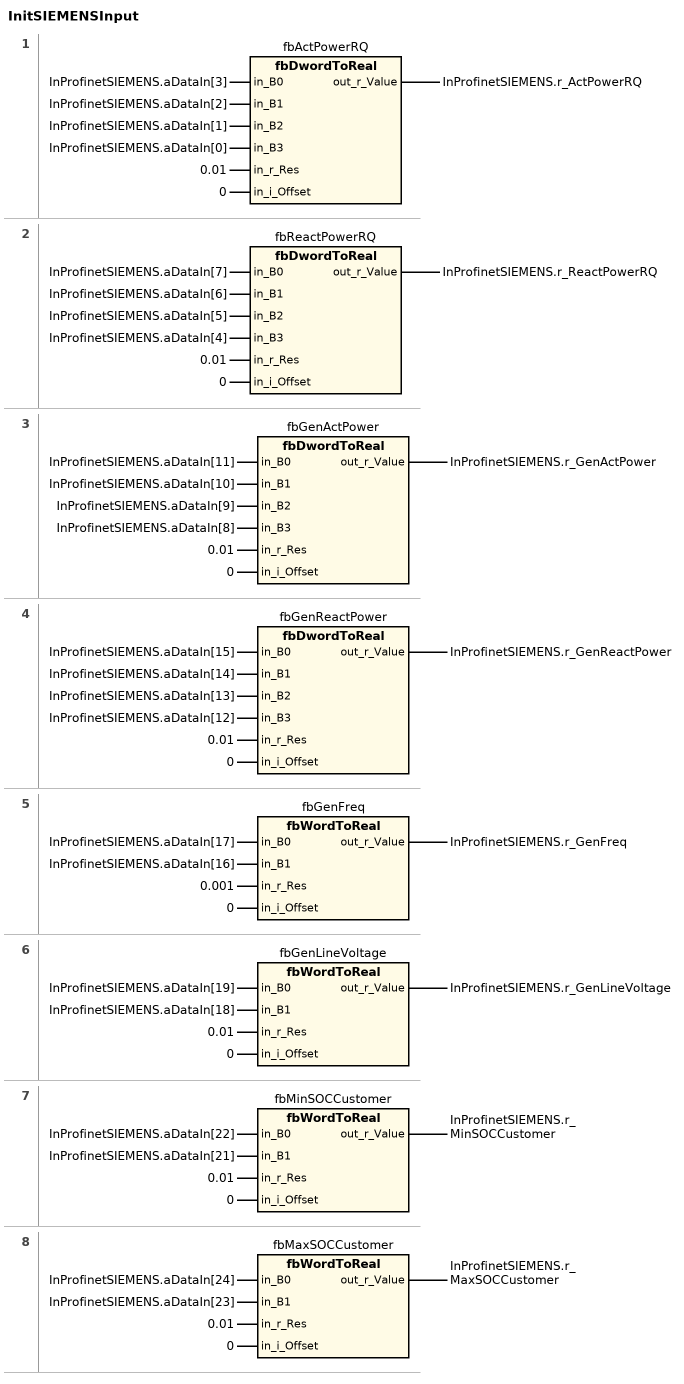
// NETWORK 1
fbActPowerRQ(
    in_B0 := InProfinetSIEMENS.aDataIn[3],
    in_B1 := InProfinetSIEMENS.aDataIn[2],
    in_B2 := InProfinetSIEMENS.aDataIn[1],
    in_B3 := InProfinetSIEMENS.aDataIn[0],
    in_r_Res := 0.01,
    in_i_Offset := 0); // fbDwordToReal
InProfinetSIEMENS.r_ActPowerRQ := fbActPowerRQ.out_r_Value;

// NETWORK 2
fbReactPowerRQ(
    in_B0 := InProfinetSIEMENS.aDataIn[7],
    in_B1 := InProfinetSIEMENS.aDataIn[6],
    in_B2 := InProfinetSIEMENS.aDataIn[5],
    in_B3 := InProfinetSIEMENS.aDataIn[4],
    in_r_Res := 0.01,
    in_i_Offset := 0); // fbDwordToReal
InProfinetSIEMENS.r_ReactPowerRQ := fbReactPowerRQ.out_r_Value;

// NETWORK 3
fbGenActPower(
    in_B0 := InProfinetSIEMENS.aDataIn[11],
    in_B1 := InProfinetSIEMENS.aDataIn[10],
    in_B2 := InProfinetSIEMENS.aDataIn[9],
    in_B3 := InProfinetSIEMENS.aDataIn[8],
    in_r_Res := 0.01,
    in_i_Offset := 0); // fbDwordToReal
InProfinetSIEMENS.r_GenActPower := fbGenActPower.out_r_Value;

// NETWORK 4
fbGenReactPower(
    in_B0 := InProfinetSIEMENS.aDataIn[15],
    in_B1 := InProfinetSIEMENS.aDataIn[14],
    in_B2 := InProfinetSIEMENS.aDataIn[13],
    in_B3 := InProfinetSIEMENS.aDataIn[12],
    in_r_Res := 0.01,
    in_i_Offset := 0); // fbDwordToReal
InProfinetSIEMENS.r_GenReactPower := fbGenReactPower.out_r_Value;

// NETWORK 5
fbGenFreq(
    in_B0 := InProfinetSIEMENS.aDataIn[17],
    in_B1 := InProfinetSIEMENS.aDataIn[16],
    in_r_Res := 0.001,
    in_i_Offset := 0); // fbWordToReal
InProfinetSIEMENS.r_GenFreq := fbGenFreq.out_r_Value;

// NETWORK 6
fbGenLineVoltage(
    in_B0 := InProfinetSIEMENS.aDataIn[19],
    in_B1 := InProfinetSIEMENS.aDataIn[18],
    in_r_Res := 0.01,
    in_i_Offset := 0); // fbWordToReal
InProfinetSIEMENS.r_GenLineVoltage := fbGenLineVoltage.out_r_Value;

// NETWORK 7
fbMinSOCCustomer(
    in_B0 := InProfinetSIEMENS.aDataIn[22],
    in_B1 := InProfinetSIEMENS.aDataIn[21],
    in_r_Res := 0.01,
    in_i_Offset := 0); // fbWordToReal
InProfinetSIEMENS.r_MinSOCCustomer := fbMinSOCCustomer.out_r_Value;

// NETWORK 8
fbMaxSOCCustomer(
    in_B0 := InProfinetSIEMENS.aDataIn[24],
    in_B1 := InProfinetSIEMENS.aDataIn[23],
    in_r_Res := 0.01,
    in_i_Offset := 0); // fbWordToReal
InProfinetSIEMENS.r_MaxSOCCustomer := fbMaxSOCCustomer.out_r_Value;

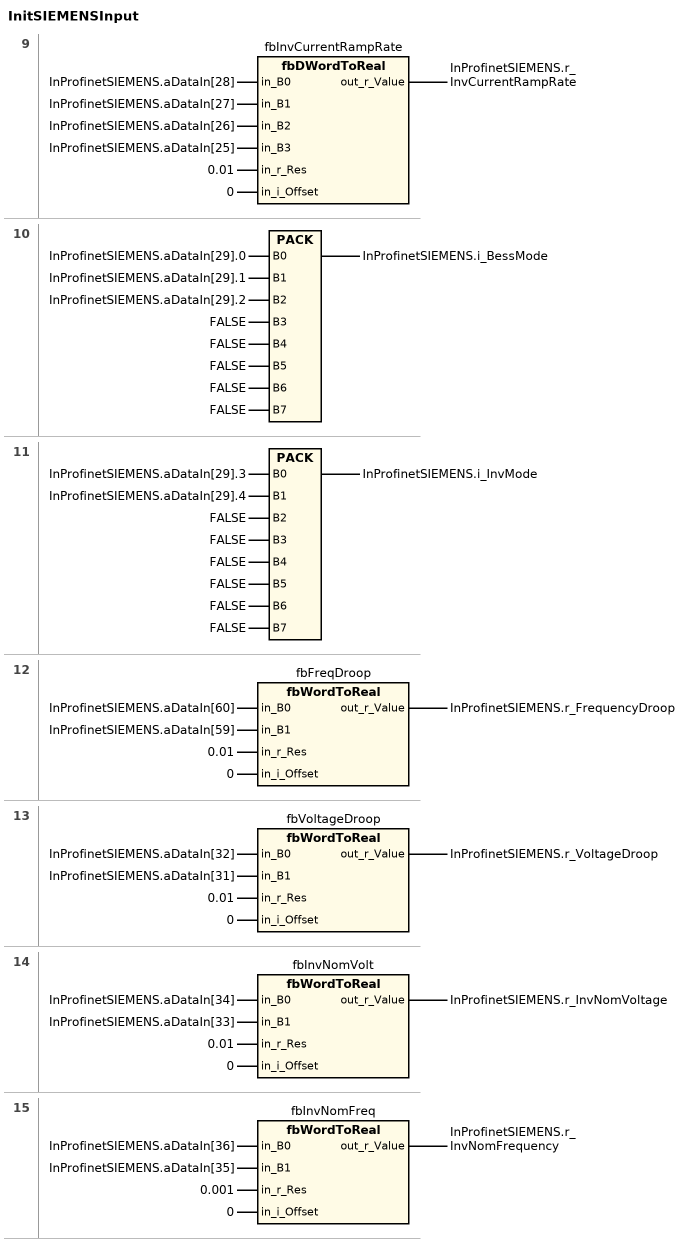
// NETWORK 9
fbInvCurrentRampRate(
    in_B0 := InProfinetSIEMENS.aDataIn[28],
    in_B1 := InProfinetSIEMENS.aDataIn[27],
    in_B2 := InProfinetSIEMENS.aDataIn[26],
    in_B3 := InProfinetSIEMENS.aDataIn[25],
    in_r_Res := 0.01,
    in_i_Offset := 0); // fbDWordToReal
InProfinetSIEMENS.r_InvCurrentRampRate := fbInvCurrentRampRate.out_r_Value;

// NETWORK 10
InProfinetSIEMENS.i_BessMode := PACK(B0 := InProfinetSIEMENS.aDataIn[29].0, B1 := InProfinetSIEMENS.aDataIn[29].1, B2 := InProfinetSIEMENS.aDataIn[29].2, B3 := FALSE, B4 := FALSE, B5 := FALSE, B6 := FALSE, B7 := FALSE);

// NETWORK 11
InProfinetSIEMENS.i_InvMode := PACK(B0 := InProfinetSIEMENS.aDataIn[29].3, B1 := InProfinetSIEMENS.aDataIn[29].4, B2 := FALSE, B3 := FALSE, B4 := FALSE, B5 := FALSE, B6 := FALSE, B7 := FALSE);

// NETWORK 12
fbFreqDroop(
    in_B0 := InProfinetSIEMENS.aDataIn[60],
    in_B1 := InProfinetSIEMENS.aDataIn[59],
    in_r_Res := 0.01,
    in_i_Offset := 0); // fbWordToReal
InProfinetSIEMENS.r_FrequencyDroop := fbFreqDroop.out_r_Value;

// NETWORK 13
fbVoltageDroop(
    in_B0 := InProfinetSIEMENS.aDataIn[32],
    in_B1 := InProfinetSIEMENS.aDataIn[31],
    in_r_Res := 0.01,
    in_i_Offset := 0); // fbWordToReal
InProfinetSIEMENS.r_VoltageDroop := fbVoltageDroop.out_r_Value;

// NETWORK 14
fbInvNomVolt(
    in_B0 := InProfinetSIEMENS.aDataIn[34],
    in_B1 := InProfinetSIEMENS.aDataIn[33],
    in_r_Res := 0.01,
    in_i_Offset := 0); // fbWordToReal
InProfinetSIEMENS.r_InvNomVoltage := fbInvNomVolt.out_r_Value;

// NETWORK 15
fbInvNomFreq(
    in_B0 := InProfinetSIEMENS.aDataIn[36],
    in_B1 := InProfinetSIEMENS.aDataIn[35],
    in_r_Res := 0.001,
    in_i_Offset := 0); // fbWordToReal
InProfinetSIEMENS.r_InvNomFrequency := fbInvNomFreq.out_r_Value;

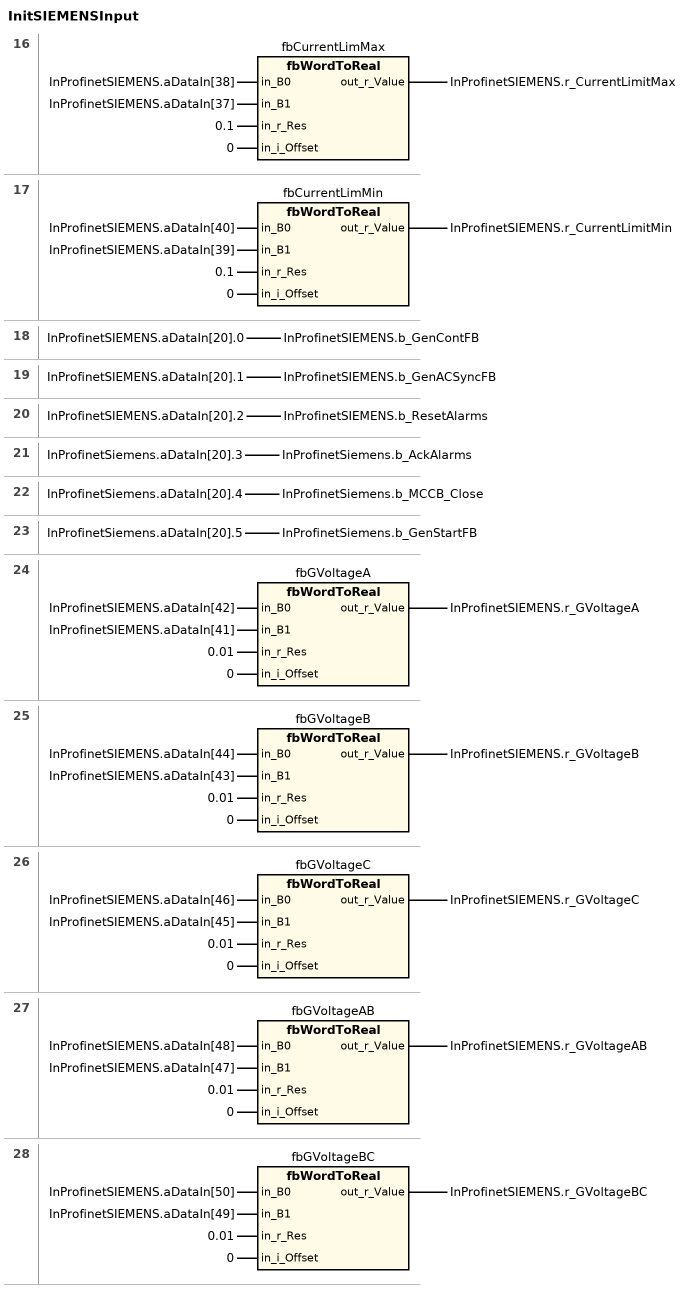
// NETWORK 16
fbCurrentLimMax(
    in_B0 := InProfinetSIEMENS.aDataIn[38],
    in_B1 := InProfinetSIEMENS.aDataIn[37],
    in_r_Res := 0.1,
    in_i_Offset := 0); // fbWordToReal
InProfinetSIEMENS.r_CurrentLimitMax := fbCurrentLimMax.out_r_Value;

// NETWORK 17
fbCurrentLimMin(
    in_B0 := InProfinetSIEMENS.aDataIn[40],
    in_B1 := InProfinetSIEMENS.aDataIn[39],
    in_r_Res := 0.1,
    in_i_Offset := 0); // fbWordToReal
InProfinetSIEMENS.r_CurrentLimitMin := fbCurrentLimMin.out_r_Value;

// NETWORK 18
InProfinetSIEMENS.b_GenContFB := InProfinetSIEMENS.aDataIn[20].0;

// NETWORK 19
InProfinetSIEMENS.b_GenACSyncFB := InProfinetSIEMENS.aDataIn[20].1;

// NETWORK 20
InProfinetSIEMENS.b_ResetAlarms := InProfinetSIEMENS.aDataIn[20].2;

// NETWORK 21
InProfinetSiemens.b_AckAlarms := InProfinetSiemens.aDataIn[20].3;

// NETWORK 22
InProfinetSiemens.b_MCCB_Close := InProfinetSiemens.aDataIn[20].4;

// NETWORK 23
InProfinetSiemens.b_GenStartFB := InProfinetSiemens.aDataIn[20].5;

// NETWORK 24
fbGVoltageA(
    in_B0 := InProfinetSIEMENS.aDataIn[42],
    in_B1 := InProfinetSIEMENS.aDataIn[41],
    in_r_Res := 0.01,
    in_i_Offset := 0); // fbWordToReal
InProfinetSIEMENS.r_GVoltageA := fbGVoltageA.out_r_Value;

// NETWORK 25
fbGVoltageB(
    in_B0 := InProfinetSIEMENS.aDataIn[44],
    in_B1 := InProfinetSIEMENS.aDataIn[43],
    in_r_Res := 0.01,
    in_i_Offset := 0); // fbWordToReal
InProfinetSIEMENS.r_GVoltageB := fbGVoltageB.out_r_Value;

// NETWORK 26
fbGVoltageC(
    in_B0 := InProfinetSIEMENS.aDataIn[46],
    in_B1 := InProfinetSIEMENS.aDataIn[45],
    in_r_Res := 0.01,
    in_i_Offset := 0); // fbWordToReal
InProfinetSIEMENS.r_GVoltageC := fbGVoltageC.out_r_Value;

// NETWORK 27
fbGVoltageAB(
    in_B0 := InProfinetSIEMENS.aDataIn[48],
    in_B1 := InProfinetSIEMENS.aDataIn[47],
    in_r_Res := 0.01,
    in_i_Offset := 0); // fbWordToReal
InProfinetSIEMENS.r_GVoltageAB := fbGVoltageAB.out_r_Value;

// NETWORK 28
fbGVoltageBC(
    in_B0 := InProfinetSIEMENS.aDataIn[50],
    in_B1 := InProfinetSIEMENS.aDataIn[49],
    in_r_Res := 0.01,
    in_i_Offset := 0); // fbWordToReal
InProfinetSIEMENS.r_GVoltageBC := fbGVoltageBC.out_r_Value;

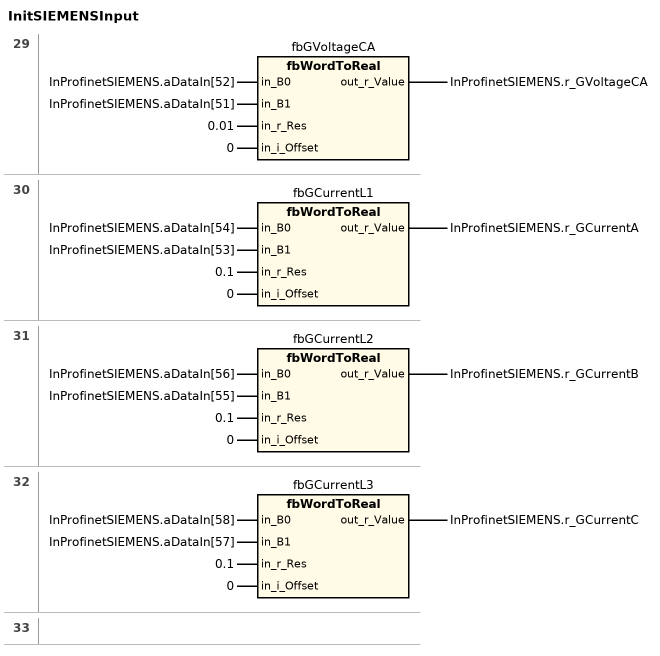
// NETWORK 29
fbGVoltageCA(
    in_B0 := InProfinetSIEMENS.aDataIn[52],
    in_B1 := InProfinetSIEMENS.aDataIn[51],
    in_r_Res := 0.01,
    in_i_Offset := 0); // fbWordToReal
InProfinetSIEMENS.r_GVoltageCA := fbGVoltageCA.out_r_Value;

// NETWORK 30
fbGCurrentL1(
    in_B0 := InProfinetSIEMENS.aDataIn[54],
    in_B1 := InProfinetSIEMENS.aDataIn[53],
    in_r_Res := 0.1,
    in_i_Offset := 0); // fbWordToReal
InProfinetSIEMENS.r_GCurrentA := fbGCurrentL1.out_r_Value;

// NETWORK 31
fbGCurrentL2(
    in_B0 := InProfinetSIEMENS.aDataIn[56],
    in_B1 := InProfinetSIEMENS.aDataIn[55],
    in_r_Res := 0.1,
    in_i_Offset := 0); // fbWordToReal
InProfinetSIEMENS.r_GCurrentB := fbGCurrentL2.out_r_Value;

// NETWORK 32
fbGCurrentL3(
    in_B0 := InProfinetSIEMENS.aDataIn[58],
    in_B1 := InProfinetSIEMENS.aDataIn[57],
    in_r_Res := 0.1,
    in_i_Offset := 0); // fbWordToReal
InProfinetSIEMENS.r_GCurrentC := fbGCurrentL3.out_r_Value;

// NETWORK 33

END_PROGRAM

// ---- POUs/ProfinetHandling/SetSiemensControlModes.TcPOU
PROGRAM SetSiemensControlModes
VAR
	i_BessMode		:INT;
	i_InvMode		:INT;
	b_Overule		: BOOL;
	TON_StorageModePulseTrigger: TON ;
	
	b_RobertTest	:BOOL;
	
	Testmode		: INT;
	
	

END_VAR

i_BessMode := InProfinetSiemens.i_BessMode;
i_InvMode  := InProfinetSiemens.i_InvMode;
IF NOT GVL.b_SiemensOverule THEN
	GVL.Gl_ShutdownIntitiatedVisu := FALSE;
	GVL.GL_UserStopVisu := FALSE;
	Safety.b_EmergencyStopVisu := FALSE;
END_IF

CASE i_BessMode OF 
	0:	//REMAIN AT CURRENT MODE
		GVL.b_ActivateSettings := FALSE;
		GVL.GL_ActivateSelectedMode := FALSE;

	1:	//SHUTDOWN
		GVL.Gl_ShutdownIntitiatedVisu := TRUE;
		
		IF (GVL.GL_StorageModeActivate OR GVL.GL_TransportModeActivate) THEN
			GVL.GL_StorageModeButtonPushed := FALSE;
		END_IF
		
	2:	// STORAGE MODE ON
		
		GVL.GL_StorageModeButtonPushed := TRUE;		;
	
		IF DigitalOutputs.b_StorageModeRelay OR GVL.GL_TransportModeActivate THEN
			OutProfinetSIEMENS.i_BessModeFB := 1;
		END_IF
		
		
		
	3: 	// TRANSPORT MODE
		//Integrated in current storage mode.
	
	4: 	// EXT CONTROL MODE
		//TO BE DONE
		
	5:	// Microgrid Mode
		GVL.GL_StorageModeButtonPushed := FALSE;
		IF (NOT DigitalInputs.b_TransferSwitchIOFF OR NOT DigitalInputs.b_TransferSwitchIIOFF) THEN
			GVL.GL_MicroGridModeButtonPushed := TRUE;
			GVL.b_ActivateSettings := TRUE;
			GVL.GL_ActivateSelectedMode := TRUE;
		END_IF
		
	6: // AFE Mode
		//TO BE DONE
		
	7: // ERROR
	Safety.b_EmergencyStopVisu	:=TRUE;
	
	IF safety.b_EmergencyStopSoftwareOK = FALSE THEN
		OutProfinetSIEMENS.i_BessModeFB := 6;
	END_IF
		
END_CASE

CASE i_InvMode	OF
	0: //REMAIN AT CURRENT MODE
	
	1: // INVERTER RUN DISABLE / OFF
		IF GVL.Gl_ShutdownIntitiatedVisu := TRUE THEN
			GVL.GL_UserStopVisu := FALSE;
		ELSE
			GVL.GL_UserStopVisu := TRUE;
		END_IF	
	
		IF GVL.Gl_ModeChangePossible := 1 THEN;
			OutProfinetSIEMENS.i_InvModeFB := 0;
		END_IF
		
	2: // ISOCHRONIOUS MODE
		GVL.i_StartPowerMode := 3;
		GVL.i_StartVoltageMode:= 2;
		
		//WHEN INVERTER MODULATION IS STOPPED, BUT MCCB STILL IN.
		IF NOT GVL.b_InverterRunning AND GVL.b_InverterReadyToOperate THEN  
			GVL.GL_ActivateSelectedMode := TRUE;
		END_IF
		
		
	3: // DROOP MODE (island)
		GVL.i_StartPowerMode := 2;
		GVL.i_StartVoltageMode:= 1;
		
		//WHEN INVERTER MODULATION IS STOPPED, BUT MCCB STILL IN.
		IF NOT GVL.b_InverterRunning AND GVL.b_InverterReadyToOperate THEN  
			GVL.GL_ActivateSelectedMode := TRUE;
		END_IF
		
	
END_CASE

//FEEDBACK SIGNAL BESS MODE
IF safety.b_EmergencyStopSoftwareOK = FALSE THEN
	OutProfinetSIEMENS.i_BessModeFB := 6;
ELSIF GVL.by_Status_ModeSequence = 17 OR GVL.by_Status_ModeSequence = 20 THEN //17 Mode off, 20 Client Setting Active
	OutProfinetSIEMENS.i_BessModeFB := 0;
ELSIF GVL.GL_StorageModeActivate THEN
	OutProfinetSIEMENS.i_BessModeFB := 1;
ELSIF GVL.b_MicroGridModeActive THEN;
	OutProfinetSIEMENS.i_BessModeFB := 4;
END_IF

// ERROR SET TO SIEMENS
IF Diagnostics.b_Error = TRUE THEN
	OutProfinetSIEMENS.i_BessModeFB := 6;
	OutProfinetSIEMENS.i_InvModeFB := 0;
END_IF


//FEEDBACK SIGNAL INVERTER MODE
IF OutProfinetInverter.i_StartPowerMode = 3 AND OutProfinetInverter.i_StartVoltageMode = 2 THEN
		OutProfinetSIEMENS.i_InvModeFB := 1;
ELSIF OutProfinetInverter.i_StartPowerMode = 2 AND OutProfinetInverter.i_StartVoltageMode = 1 THEN
		OutProfinetSIEMENS.i_InvModeFB := 2;
END_IF

END_PROGRAM

// ---- POUs/ProfinetHandling/SetSIEMENSOutput.TcPOU
PROGRAM SetSIEMENSOutput
VAR
	fbSocCustomerLowLimit		: fbRealToWord;
	fbSocCustomerHighLimit		: fbRealToWord;
	fbCalculatedSOC				: fbRealToWord;
	fbSOH						: fbRealToWord;
	fbMaxChargeCurrent			: fbRealToWord;
	fbMaxDischargeCurrent		: fbRealToWord;
	fbCurrentLimitMax			: fbRealToWord;
	fbCurrentLimitMin			: fbRealToWord;
	fbActiveCurrent				: fbRealToDWord;
	fbReactiveCurrent			: fbRealToDWord;
	fbVoltageA					: fbRealToWord;
	fbVoltageB					: fbRealToWord;
	fbVoltageC					: fbRealToWord;
	fbVoltageAB					: fbRealToWord;
	fbVoltageBC					: fbRealToWord;
	fbVoltageCA					: fbRealToWord;
	fbCurrentA					: fbRealToDWord;
	fbCurrentB					: fbRealToDWord;
	fbCurrentC					: fbRealToDWord;
	fbCurrentN					: fbRealToDWord;
	fbLineVoltage				: fbRealToWord;
	fbSupplyVoltage				: fbRealToWord;
	fbLineFreq					: fbRealToWord;
	fbSupplyFreq				: fbRealToWord;
	fbTotalUsedEnergy			: fbRealToDWord;
	fbTemperatureBatteryCompartment		: fbRealToWord;
	fbTemperatureElectricalCompartment		: fbRealToWord;
	fbMinCellTemperature		: fbRealToWord;
	fbMaxCellTemperature		: fbRealToWord;
	fbAvgCellTemperature		: fbRealToWord;
	fbSOCUPS1		: fbRealToWord;
	fbSOCRemainingTimeUPS1		: fbRealToWord;
	fbTransformerTemp			: fbRealToWord;
	fbInverterTemp			: fbRealToWord;
	fbActPowerPQMeter			: fbRealToWord;
	fbReactPowerPQMeter			: fbRealToWord;
	
			
	fbDCLinkVoltage		: fbRealToDWord;
	fbDCLinkCurrent		: fbRealToDWord;
	fbMinCellVoltage		: fbRealToWord;
	fbMaxCellVoltage		: fbRealToWord;
	fbAvgCellVoltage		: fbRealToWord;
	
	b_GenACSyncPerm: BOOL := TRUE;
	b_Spare: BOOL;
END_VAR


fbSocCustomerLowLimit(in_r_Value:= GVL.r_SocCustomerLowLimitVISU,in_r_Res:= 0.01, in_i_Offset:= 0,out_B0=> OutProfinetSIEMENS.aDataOut[1], out_B1=> OutProfinetSIEMENS.aDataOut[0]);
fbSocCustomerHighLimit(in_r_Value:= GVL.r_SocCustomerHighLimitVISU,in_r_Res:= 0.01, in_i_Offset:= 0,out_B0=> OutProfinetSIEMENS.aDataOut[3], out_B1=> OutProfinetSIEMENS.aDataOut[2]);
fbCalculatedSOC(in_r_Value:= GVL.lr_CalculatedSOC,in_r_Res:= 0.01, in_i_Offset:= 0,out_B0=> OutProfinetSIEMENS.aDataOut[5], out_B1=> OutProfinetSIEMENS.aDataOut[4]);
fbSOH(in_r_Value:= InCanBMS.lr_SOH,in_r_Res:= 0.01, in_i_Offset:= 0,out_B0=> OutProfinetSIEMENS.aDataOut[7], out_B1=> OutProfinetSIEMENS.aDataOut[6]);
fbMaxChargeCurrent(in_r_Value:= GVL.r_MaxChargeCurrentAC,in_r_Res:= 0.01, in_i_Offset:= 0,out_B0=> OutProfinetSIEMENS.aDataOut[9], out_B1=> OutProfinetSIEMENS.aDataOut[8]);
fbMaxDischargeCurrent(in_r_Value:= GVL.r_MaxDischargeCurrentAC,in_r_Res:= 0.01, in_i_Offset:= 0,out_B0=> OutProfinetSIEMENS.aDataOut[11], out_B1=> OutProfinetSIEMENS.aDataOut[10]);
fbActiveCurrent(in_r_Value:= GVL.r_InvActiveCurrent,in_r_Res:= 0.01, in_i_Offset:= 0,out_B0=> OutProfinetSIEMENS.aDataOut[15], out_B1=> OutProfinetSIEMENS.aDataOut[14], out_B2=> OutProfinetSIEMENS.aDataOut[13], out_B3=> OutProfinetSIEMENS.aDataOut[12]);
fbReactiveCurrent(in_r_Value:= GVL.r_InvReactiveCurrent,in_r_Res:= 0.01, in_i_Offset:= 0,out_B0=> OutProfinetSIEMENS.aDataOut[19], out_B1=> OutProfinetSIEMENS.aDataOut[18], out_B2=> OutProfinetSIEMENS.aDataOut[17], out_B3=> OutProfinetSIEMENS.aDataOut[16]);
OutProfinetSIEMENS.aDataOut[20] := REAL_TO_BYTE(PowerMonitoringTCP.r_ActivePowerFactor/0.01);
fbVoltageA(in_r_Value:= PowerMonitoringTCP.r_VoltageA_N,in_r_Res:= 0.01, in_i_Offset:= 0,out_B0=> OutProfinetSIEMENS.aDataOut[22], out_B1=> OutProfinetSIEMENS.aDataOut[21]);
fbVoltageB(in_r_Value:= PowerMonitoringTCP.r_VoltageB_N,in_r_Res:= 0.01, in_i_Offset:= 0,out_B0=> OutProfinetSIEMENS.aDataOut[24], out_B1=> OutProfinetSIEMENS.aDataOut[23]);
fbVoltageC(in_r_Value:= PowerMonitoringTCP.r_VoltageC_N,in_r_Res:= 0.01, in_i_Offset:= 0,out_B0=> OutProfinetSIEMENS.aDataOut[26], out_B1=> OutProfinetSIEMENS.aDataOut[25]);
fbVoltageAB(in_r_Value:= PowerMonitoringTCP.r_VoltageAB,in_r_Res:= 0.01, in_i_Offset:= 0,out_B0=> OutProfinetSIEMENS.aDataOut[28], out_B1=> OutProfinetSIEMENS.aDataOut[27]);
fbVoltageBC(in_r_Value:= PowerMonitoringTCP.r_VoltageBC,in_r_Res:= 0.01, in_i_Offset:= 0,out_B0=> OutProfinetSIEMENS.aDataOut[30], out_B1=> OutProfinetSIEMENS.aDataOut[29]);
fbVoltageCA(in_r_Value:= PowerMonitoringTCP.r_VoltageCA,in_r_Res:= 0.01, in_i_Offset:= 0,out_B0=> OutProfinetSIEMENS.aDataOut[32], out_B1=> OutProfinetSIEMENS.aDataOut[31]);
fbCurrentA(in_r_Value:= PowerMonitoringTCP.r_CurrentA,in_r_Res:= 0.01, in_i_Offset:= 0,out_B0=> OutProfinetSIEMENS.aDataOut[36], out_B1=> OutProfinetSIEMENS.aDataOut[35], out_B2=> OutProfinetSIEMENS.aDataOut[34], out_B3=> OutProfinetSIEMENS.aDataOut[33]);
fbCurrentB(in_r_Value:= PowerMonitoringTCP.r_CurrentB,in_r_Res:= 0.01, in_i_Offset:= 0,out_B0=> OutProfinetSIEMENS.aDataOut[40], out_B1=> OutProfinetSIEMENS.aDataOut[39], out_B2=> OutProfinetSIEMENS.aDataOut[38], out_B3=> OutProfinetSIEMENS.aDataOut[37]);
fbCurrentC(in_r_Value:= PowerMonitoringTCP.r_CurrentC,in_r_Res:= 0.01, in_i_Offset:= 0,out_B0=> OutProfinetSIEMENS.aDataOut[44], out_B1=> OutProfinetSIEMENS.aDataOut[43], out_B2=> OutProfinetSIEMENS.aDataOut[42], out_B3=> OutProfinetSIEMENS.aDataOut[41]);
fbCurrentN(in_r_Value:= PowerMonitoringTCP.r_CurrentN,in_r_Res:= 0.01, in_i_Offset:= 0,out_B0=> OutProfinetSIEMENS.aDataOut[48], out_B1=> OutProfinetSIEMENS.aDataOut[47], out_B2=> OutProfinetSIEMENS.aDataOut[46], out_B3=> OutProfinetSIEMENS.aDataOut[45]);
fbLineVoltage(in_r_Value:= GVL.r_InvLineVoltageD7,in_r_Res:= 0.01, in_i_Offset:= 0,out_B0=> OutProfinetSIEMENS.aDataOut[50], out_B1=> OutProfinetSIEMENS.aDataOut[49]);
fbLineFreq(in_r_Value:= GVL.r_InvLineFrequencyD7,in_r_Res:= 0.01, in_i_Offset:= 0,out_B0=> OutProfinetSIEMENS.aDataOut[52], out_B1=> OutProfinetSIEMENS.aDataOut[51]);
fbTotalUsedEnergy(in_r_Value:= UDINT_TO_REAL(InCanBMS.usi_TotalUsedEnergy),in_r_Res:= 0.01, in_i_Offset:= 0,out_B0=> OutProfinetSIEMENS.aDataOut[56], out_B1=> OutProfinetSIEMENS.aDataOut[55], out_B2=> OutProfinetSIEMENS.aDataOut[54], out_B3=> OutProfinetSIEMENS.aDataOut[53]);
fbTemperatureBatteryCompartment(in_r_Value:= AI.r_TemperatureBatteryCompartment,in_r_Res:= 0.01, in_i_Offset:= 0,out_B0=> OutProfinetSIEMENS.aDataOut[58], out_B1=> OutProfinetSIEMENS.aDataOut[57]);
fbTemperatureElectricalCompartment(in_r_Value:= AI.r_TemperatureElectricalCompartment,in_r_Res:= 0.01, in_i_Offset:= 0,out_B0=> OutProfinetSIEMENS.aDataOut[60], out_B1=> OutProfinetSIEMENS.aDataOut[59]);
fbMinCellTemperature(in_r_Value:= LREAL_TO_REAL(InCanBMS.lr_MinCellTemperature),in_r_Res:= 0.01, in_i_Offset:= 0,out_B0=> OutProfinetSIEMENS.aDataOut[62], out_B1=> OutProfinetSIEMENS.aDataOut[61]);
fbMaxCellTemperature(in_r_Value:= LREAL_TO_REAL(InCanBMS.lr_MaxCellTemperature),in_r_Res:= 0.01, in_i_Offset:= 0,out_B0=> OutProfinetSIEMENS.aDataOut[64], out_B1=> OutProfinetSIEMENS.aDataOut[63]);
fbAvgCellTemperature(in_r_Value:= LREAL_TO_REAL(InCanBMS.lr_AvgCellTemperature),in_r_Res:= 0.01, in_i_Offset:= 0,out_B0=> OutProfinetSIEMENS.aDataOut[66], out_B1=> OutProfinetSIEMENS.aDataOut[65]);
fbSOCUPS1(in_r_Value:= GVL.r_UPSBatSoC,in_r_Res:= 0.01, in_i_Offset:= 0,out_B0=> OutProfinetSIEMENS.aDataOut[68], out_B1=> OutProfinetSIEMENS.aDataOut[67]);
fbSOCRemainingTimeUPS1(in_r_Value:= GVL.r_UPSTimeRemaining,in_r_Res:= 0.01, in_i_Offset:= 0,out_B0=> OutProfinetSIEMENS.aDataOut[70], out_B1=> OutProfinetSIEMENS.aDataOut[69]);
OutProfinetSIEMENS.aDataOut[71] := REAL_TO_BYTE(InProfinetUPS.di_StatusPSU1/1);
fbDCLinkVoltage(in_r_Value:= GVL.r_DCLinkVoltage,in_r_Res:= 0.01, in_i_Offset:= 0,out_B0=> OutProfinetSIEMENS.aDataOut[75], out_B1=> OutProfinetSIEMENS.aDataOut[74], out_B2=> OutProfinetSIEMENS.aDataOut[73], out_B3=> OutProfinetSIEMENS.aDataOut[72]);
fbDCLinkCurrent(in_r_Value:= GVL.r_DCLinkCurrent,in_r_Res:= 0.01, in_i_Offset:= 0,out_B0=> OutProfinetSIEMENS.aDataOut[79], out_B1=> OutProfinetSIEMENS.aDataOut[78], out_B2=> OutProfinetSIEMENS.aDataOut[77], out_B3=> OutProfinetSIEMENS.aDataOut[76]);
fbMinCellVoltage(in_r_Value:= UINT_TO_REAL(InCanBMS.ui_MinCellVoltage),in_r_Res:= 1, in_i_Offset:= 0,out_B0=> OutProfinetSIEMENS.aDataOut[81], out_B1=> OutProfinetSIEMENS.aDataOut[80]);
fbMaxCellVoltage(in_r_Value:= UINT_TO_REAL(InCanBMS.ui_MaxCellVoltage),in_r_Res:= 1, in_i_Offset:= 0,out_B0=> OutProfinetSIEMENS.aDataOut[83], out_B1=> OutProfinetSIEMENS.aDataOut[82]);
fbAvgCellVoltage(in_r_Value:= UINT_TO_REAL(InCanBMS.ui_AvgCellVoltage),in_r_Res:= 1, in_i_Offset:= 0,out_B0=> OutProfinetSIEMENS.aDataOut[85], out_B1=> OutProfinetSIEMENS.aDataOut[84]);
fbCurrentLimitMax(in_r_Value:= OutProfinetInverter.i_CurrentlimitMax,in_r_Res:= 0.1, in_i_Offset:= 0,out_B0=> OutProfinetSIEMENS.aDataOut[89], out_B1=> OutProfinetSIEMENS.aDataOut[88]);
fbCurrentLimitMin(in_r_Value:= OutProfinetInverter.i_CurrentlimitMax,in_r_Res:= 0.1, in_i_Offset:= 0,out_B0=> OutProfinetSIEMENS.aDataOut[91], out_B1=> OutProfinetSIEMENS.aDataOut[90]);
OutProfinetSIEMENS.aDataOut[129]:= GVL.by_Status_ModeSequence;
fbSupplyFreq(in_r_Value:= GVL.r_InvSupplyFrequency,in_r_Res:= 0.01, in_i_Offset:= 0,out_B0=> OutProfinetSIEMENS.aDataOut[131], out_B1=> OutProfinetSIEMENS.aDataOut[130]);
fbSupplyVoltage(in_r_Value:= GVL.r_InvSupplyVoltage,in_r_Res:= 0.01, in_i_Offset:= 0,out_B0=> OutProfinetSIEMENS.aDataOut[133], out_B1=> OutProfinetSIEMENS.aDataOut[132]);
fbTransformerTemp(in_r_Value:= AI.r_TemperatureTransformer, in_r_Res:=0.1, in_i_Offset:=0, out_B0=> OutProfinetSIEMENS.aDataOut[135], out_B1=> OutProfinetSIEMENS.aDataOut[134]);
fbInverterTemp(in_r_Value:= GVL.r_InvTemperature, in_r_Res:=0.1, in_i_Offset:=0, out_B0=> OutProfinetSIEMENS.aDataOut[137], out_B1=> OutProfinetSIEMENS.aDataOut[136]);
fbActPowerPQMeter(in_r_Value:= PowerMonitoringTCP.r_ActivePower, in_r_Res:=0.01, in_i_Offset:=0, out_B0=> OutProfinetSIEMENS.aDataOut[139], out_B1=> OutProfinetSIEMENS.aDataOut[138]); 
fbReactPowerPQMeter(in_r_Value:= PowerMonitoringTCP.r_ReactivePower, in_r_Res:=0.01, in_i_Offset:=0, out_B0=> OutProfinetSIEMENS.aDataOut[141], out_B1=> OutProfinetSIEMENS.aDataOut[140]); 
//Feedback Signals



// Diagnostics
OutProfinetSIEMENS.aDataOut[86].0 := Diagnostics.b_ACRotationFault;
OutProfinetSIEMENS.aDataOut[86].1 := b_GenACSyncPerm;
OutProfinetSIEMENS.aDataOut[86].2 := DigitalInputs.b_AirconditioningOK;
OutProfinetSIEMENS.aDataOut[86].3 := DigitalInputs.b_TransferSwitchIOFF;
OutProfinetSIEMENS.aDataOut[86].4 := DigitalInputs.b_TransferSwitchIIOFF;
OutprofinetSIEMENS.aDataOut[86].5 := GVL.b_MCCB_Active;
OutprofinetSIEMENS.aDataOut[86].6 := DigitalInputs.b_DisconnectorIOFF;
OutprofinetSIEMENS.aDataOut[86].7 := DigitalInputs.b_DisconnectorIIOFF;
OutprofinetSIEMENS.aDataOut[87].1 := GVL.b_GenStartStopEnable;
OutProfinetSIEMENS.aDataOut[100].0 := Diagnostics.b_DoorElectricalCompartmentOpen;
OutProfinetSIEMENS.aDataOut[100].1 := Diagnostics.b_AircoTurnedOff;
OutProfinetSIEMENS.aDataOut[100].2 := Diagnostics.b_Door1BatteryCompartmentOpen;
OutProfinetSIEMENS.aDataOut[100].3 := Diagnostics.b_PowerSupplyFusesNOK          ;
OutProfinetSIEMENS.aDataOut[100].4 := Diagnostics.b_PowerSupplyHVFusesNOK        ;
OutProfinetSIEMENS.aDataOut[100].5 := Diagnostics.b_PowerSupply400VACDanfossNOK  ;
OutProfinetSIEMENS.aDataOut[100].6 := Diagnostics.b_PowerSupply400VACNOK         ;
OutProfinetSIEMENS.aDataOut[100].7 := Diagnostics.b_PowerSupply230VACNOK         ;
OutProfinetSIEMENS.aDataOut[101].0 := Diagnostics.b_PowerSupply3F400VACNOK       ;
OutProfinetSIEMENS.aDataOut[101].1 := Diagnostics.b_PowerInlet3x400VACNOK        ;
OutProfinetSIEMENS.aDataOut[101].2 := Diagnostics.b_FireDetected;
OutProfinetSIEMENS.aDataOut[101].3 := Diagnostics.b_DriveTripped;
OutProfinetSIEMENS.aDataOut[101].4 := Diagnostics.b_TemperatureElectricalHigh;
OutProfinetSIEMENS.aDataOut[101].5 := Diagnostics.b_HumidityElectricalHigh;
OutProfinetSIEMENS.aDataOut[101].6 := Diagnostics.b_TemperatureBatteryHigh;
OutProfinetSIEMENS.aDataOut[101].7 := Diagnostics.b_HumidityBatteryHigh;
OutProfinetSIEMENS.aDataOut[102].0 := Diagnostics.b_HumidityElectricalTooHigh;
OutProfinetSIEMENS.aDataOut[102].1 := Diagnostics.b_TemperatureElectricalTooHigh;
OutProfinetSIEMENS.aDataOut[102].2 := Diagnostics.b_HumidityBatteryTooHigh;
OutProfinetSIEMENS.aDataOut[102].3 := Diagnostics.b_TemperatureBatteryTooHigh;
OutProfinetSIEMENS.aDataOut[102].4 := Diagnostics.b_Spare;
OutProfinetSIEMENS.aDataOut[102].5 := Diagnostics.b_String1Absent;
OutProfinetSIEMENS.aDataOut[102].6 := Diagnostics.b_String2Absent;
OutProfinetSIEMENS.aDataOut[102].7 := Diagnostics.b_String3Absent;
OutProfinetSIEMENS.aDataOut[103].0 := Diagnostics.b_String4Absent;
OutProfinetSIEMENS.aDataOut[103].1 := Diagnostics.b_String5Absent;
OutProfinetSIEMENS.aDataOut[103].2 := Diagnostics.b_String6Absent;
OutProfinetSIEMENS.aDataOut[103].3 := Diagnostics.b_ALOCellTempLow;
OutProfinetSIEMENS.aDataOut[103].4 := Diagnostics.b_ALOCellTempHigh;
OutProfinetSIEMENS.aDataOut[103].5 := Diagnostics.b_AVGCellTempLow;
OutProfinetSIEMENS.aDataOut[103].6 := Diagnostics.b_AVGCellTempHigh;
OutProfinetSIEMENS.aDataOut[103].7 := Diagnostics.b_ALOCellVoltageLow;
OutProfinetSIEMENS.aDataOut[104].0 := Diagnostics.b_ALOCellVoltageHigh;
OutProfinetSIEMENS.aDataOut[104].1 := Diagnostics.b_AVGCellVoltageLow;
OutProfinetSIEMENS.aDataOut[104].2 := Diagnostics.b_AVGCellVoltageHigh;
OutProfinetSIEMENS.aDataOut[104].3 := Diagnostics.b_OverCurrent10s;
OutProfinetSIEMENS.aDataOut[104].4 := Diagnostics.b_SOCLow;
OutProfinetSIEMENS.aDataOut[104].5 := Diagnostics.b_EmergencyError;
OutProfinetSIEMENS.aDataOut[104].6 := Diagnostics.b_CellCapacityTooLow;
OutProfinetSIEMENS.aDataOut[104].7 := Diagnostics.b_CellCapacityTooHigh;
OutProfinetSIEMENS.aDataOut[105].0 := Diagnostics.b_ALOCellTempTooLow;
OutProfinetSIEMENS.aDataOut[105].1 := Diagnostics.b_ALOCellTempTooHigh;
OutProfinetSIEMENS.aDataOut[105].2 := Diagnostics.b_AVGCellTempTooLow;
OutProfinetSIEMENS.aDataOut[105].3 := Diagnostics.b_AVGCellTempTooHigh;
OutProfinetSIEMENS.aDataOut[105].4 := Diagnostics.b_ALOCellVoltageTooLow;
OutProfinetSIEMENS.aDataOut[105].5 := Diagnostics.b_ALOCellVoltageTooHigh;
OutProfinetSIEMENS.aDataOut[105].6 := Diagnostics.b_AVGCellVoltageTooLow;
OutProfinetSIEMENS.aDataOut[105].7 := Diagnostics.b_AVGCellVoltageTooHigh;
OutProfinetSIEMENS.aDataOut[106].0 := Diagnostics.b_Overcurrent;
OutProfinetSIEMENS.aDataOut[106].1 := Diagnostics.b_SystemVoltageTooHigh;
OutProfinetSIEMENS.aDataOut[106].2 := Diagnostics.b_SystemVoltageTooLow;
OutProfinetSIEMENS.aDataOut[106].3 := Diagnostics.b_SOCTooLow;
OutProfinetSIEMENS.aDataOut[106].4 := Diagnostics.b_SOCToohigh;
OutProfinetSIEMENS.aDataOut[106].5 := Diagnostics.b_BatteryLimitsExceeded;
OutProfinetSIEMENS.aDataOut[106].6 := Diagnostics.b_BMSErrorState;
OutProfinetSIEMENS.aDataOut[106].7 := Diagnostics.b_InverterFault;
OutProfinetSIEMENS.aDataOut[107].0 := Diagnostics.b_CBControlNotOK;
OutProfinetSIEMENS.aDataOut[107].1 := Diagnostics.b_WarningInverter;
OutProfinetSIEMENS.aDataOut[107].2 := Diagnostics.b_DCAboveLimit;
OutProfinetSIEMENS.aDataOut[107].3 := Diagnostics.b_F1OverCurrent;
OutProfinetSIEMENS.aDataOut[107].4 := Diagnostics.b_F2OverVoltage;
OutProfinetSIEMENS.aDataOut[107].5 := Diagnostics.b_F9UnderVoltage;
OutProfinetSIEMENS.aDataOut[107].6 := Diagnostics.b_F91ShortCircuit;
OutProfinetSIEMENS.aDataOut[107].7 := Diagnostics.b_F3EarthFault;
OutProfinetSIEMENS.aDataOut[108].0 := Diagnostics.b_F14UnitOverTemperature;
OutProfinetSIEMENS.aDataOut[108].1 := Diagnostics.b_F56TemperatureFault;
OutProfinetSIEMENS.aDataOut[108].2 := Diagnostics.b_F10LineSynchFault;
OutProfinetSIEMENS.aDataOut[108].3 := Diagnostics.b_F52KeypadOCCommFault;
OutProfinetSIEMENS.aDataOut[108].4 := Diagnostics.b_F53FieldbusFault;
OutProfinetSIEMENS.aDataOut[108].5 := Diagnostics.b_F59SystembusFault;
OutProfinetSIEMENS.aDataOut[108].6 := Diagnostics.b_F54SlotCommunicationFault;
OutProfinetSIEMENS.aDataOut[108].7 := Diagnostics.b_F50Meas4mAFault;
OutProfinetSIEMENS.aDataOut[109].0 := Diagnostics.b_AlarmDeviceReady;
OutProfinetSIEMENS.aDataOut[109].1 := Diagnostics.b_AlarmCurrentA ;
OutProfinetSIEMENS.aDataOut[109].2 := Diagnostics.b_AlarmCurrentB ;
OutProfinetSIEMENS.aDataOut[109].3 := Diagnostics.b_AlarmCurrentC ;
OutProfinetSIEMENS.aDataOut[109].4 := Diagnostics.b_AlarmVoltageAB;
OutProfinetSIEMENS.aDataOut[109].5 := Diagnostics.b_AlarmVoltageBC;
OutProfinetSIEMENS.aDataOut[109].6 := Diagnostics.b_AlarmVoltageCA;
OutProfinetSIEMENS.aDataOut[109].7 := Diagnostics.b_AlarmActivePower;
OutProfinetSIEMENS.aDataOut[110].0 := Diagnostics.b_AlarmReactivePower;
OutProfinetSIEMENS.aDataOut[110].1 := Diagnostics.b_AlarmApparentPower;
OutProfinetSIEMENS.aDataOut[110].2 := Diagnostics.b_AlarmActivePowerFactor;
OutProfinetSIEMENS.aDataOut[110].3 := Diagnostics.b_AlarmFrequency;
OutProfinetSIEMENS.aDataOut[110].4 := Diagnostics.b_AlarmDemandActiveEnergy;
OutProfinetSIEMENS.aDataOut[110].5 := Diagnostics.b_AlarmSupplyActiveEnergy;
OutProfinetSIEMENS.aDataOut[110].6 := Diagnostics.b_Insulation1Alarm ;
OutProfinetSIEMENS.aDataOut[110].7 := Diagnostics.b_Insulation2Alarm ;
OutProfinetSIEMENS.aDataOut[111].0 := Diagnostics.b_ConnectionFault ;
OutProfinetSIEMENS.aDataOut[111].1 := Diagnostics.b_DCMinAlarm ;
OutProfinetSIEMENS.aDataOut[111].2 := Diagnostics.b_DCPlusAlarm ;
OutProfinetSIEMENS.aDataOut[111].3 := Diagnostics.b_SymmectricalAlarm;
OutProfinetSIEMENS.aDataOut[111].4 := Diagnostics.b_DeviceError ;
OutProfinetSIEMENS.aDataOut[111].5 := Diagnostics.b_CommonAlarm;
OutProfinetSIEMENS.aDataOut[111].6 := Diagnostics.b_MeasurementAlarm;
OutProfinetSIEMENS.aDataOut[111].7 := Diagnostics.b_DeviceInactive;
OutProfinetSIEMENS.aDataOut[112].0 := Diagnostics.b_DCOffsetAlarm ;
OutProfinetSIEMENS.aDataOut[112].1 := Diagnostics.b_CommonEDSAlarm;
OutProfinetSIEMENS.aDataOut[112].2 := Diagnostics.b_PGHPulseAlarm;
OutProfinetSIEMENS.aDataOut[112].3 := Diagnostics.b_ISOnetMeasurementAlarm;
OutProfinetSIEMENS.aDataOut[112].4 := Diagnostics.b_PGHActiveAlarm;
OutProfinetSIEMENS.aDataOut[112].5 := Diagnostics.b_CommunicationError;
OutProfinetSIEMENS.aDataOut[112].6 := Diagnostics.b_AlarmSoftwareVersion;
OutProfinetSIEMENS.aDataOut[112].7 := Diagnostics.b_AlarmIsolationDeviceReady;
OutProfinetSIEMENS.aDataOut[113].0 := Diagnostics.b_AlarmNumberEquipments;
OutProfinetSIEMENS.aDataOut[113].1 := Diagnostics.b_AlarmDigitalOutput1;
OutProfinetSIEMENS.aDataOut[113].2 := Diagnostics.b_AlarmDigitalOutput2;
OutProfinetSIEMENS.aDataOut[113].3 := Diagnostics.b_AlarmBuzzerFunctional;
OutProfinetSIEMENS.aDataOut[113].4 := Diagnostics.b_AlarmRelayOperationMode;
OutProfinetSIEMENS.aDataOut[113].5 := Diagnostics.b_AlarmRelay2OperationMode;
OutProfinetSIEMENS.aDataOut[113].6 := Diagnostics.b_AlarmResponseValue1;
OutProfinetSIEMENS.aDataOut[113].7 := Diagnostics.b_AlarmResponseValue2;
OutProfinetSIEMENS.aDataOut[114].0 := Diagnostics.b_AlarmSystemType;
OutProfinetSIEMENS.aDataOut[114].1 := Diagnostics.b_AlarmProfile;
OutProfinetSIEMENS.aDataOut[114].2 := Diagnostics.b_AlarmInsulationResistance;
OutProfinetSIEMENS.aDataOut[114].3 := Diagnostics.b_AlarmTestStatus;
OutProfinetSIEMENS.aDataOut[114].4 := Diagnostics.b_AlarmAlarmStatus;
OutProfinetSIEMENS.aDataOut[114].5 := Diagnostics.b_AlarmRange;
OutProfinetSIEMENS.aDataOut[114].6 := Diagnostics.b_AlarmUnit;
OutProfinetSIEMENS.aDataOut[114].7 := Diagnostics.b_AlarmInsulationResistance2;
OutProfinetSIEMENS.aDataOut[115].0 := Diagnostics.b_AlarmVoltageL1L3;
OutProfinetSIEMENS.aDataOut[115].1 := Diagnostics.b_AlarmIOState;
OutProfinetSIEMENS.aDataOut[115].2 := Diagnostics.b_AlarmAlarmStatus2;
OutProfinetSIEMENS.aDataOut[115].3 := Diagnostics.b_ResetAlarm;
OutProfinetSIEMENS.aDataOut[115].4 := Diagnostics.b_Error;
OutProfinetSIEMENS.aDataOut[115].5 := Diagnostics.b_Warning;
OutProfinetSIEMENS.aDataOut[115].6 := Diagnostics.b_ClearHistory;
OutProfinetSIEMENS.aDataOut[115].7 := Diagnostics.b_NormalShutdown ;
OutProfinetSIEMENS.aDataOut[116].0 := Diagnostics.b_EmergencyShutdown ;
OutProfinetSIEMENS.aDataOut[116].1 := Diagnostics.b_SelectModus;
OutProfinetSIEMENS.aDataOut[116].2 := Diagnostics.b_SelectSubModus;
OutProfinetSIEMENS.aDataOut[116].3 := Diagnostics.b_ActivatePowerSettings;
OutProfinetSIEMENS.aDataOut[116].4 := Diagnostics.b_EmergencyStopSafety;
OutProfinetSIEMENS.aDataOut[116].5 := Diagnostics.b_EmergencyStopDelayedSafety;
OutProfinetSIEMENS.aDataOut[116].6 := Diagnostics.b_EmergencyStopChannel1 ;
OutProfinetSIEMENS.aDataOut[116].7 := Diagnostics.b_EmergencyStopChannel2 ;
OutProfinetSIEMENS.aDataOut[117].0 := Diagnostics.b_IsolationWarningDC ;
OutProfinetSIEMENS.aDataOut[117].1 := Diagnostics.b_IsolationErrorDC ;
OutProfinetSIEMENS.aDataOut[117].2 := Diagnostics.b_IsolationWarningAC ;
OutProfinetSIEMENS.aDataOut[117].3 := Diagnostics.b_IsolationErrorAC;
OutProfinetSIEMENS.aDataOut[117].4 := Diagnostics.b_EmergencyShutdownSoftware;
OutProfinetSIEMENS.aDataOut[117].5 := Diagnostics.b_EmergencyOpenBMS;
OutProfinetSIEMENS.aDataOut[117].6 := Diagnostics.b_InverterWatchDogError;

OutProfinetSIEMENS.aDataOut[117].7 := Diagnostics.b_TemperatureElectricalTooHigh;
OutProfinetSIEMENS.aDataOut[118].0 := Diagnostics.b_TemperatureBatteryTooHigh;
OutProfinetSIEMENS.aDataOut[118].1 := Diagnostics.b_HumidityElectricalTooHigh;
OutProfinetSIEMENS.aDataOut[118].2 := Diagnostics.b_HumidityBatteryTooHigh;

OutProfinetSIEMENS.aDataOut[118].3 := Diagnostics.b_BmsStateNok;
OutProfinetSIEMENS.aDataOut[118].4 := Diagnostics.b_FireDetectionSystemFault;
OutProfinetSIEMENS.aDataOut[118].5 := Diagnostics.b_DoorInverterCabinetOpen;
OutProfinetSIEMENS.aDataOut[118].6 := Diagnostics.b_TransportModeConditionsNOK;
OutProfinetSIEMENS.aDataOut[118].7 := Diagnostics.b_EdmErrorPowerSupplyRelais;
OutProfinetSIEMENS.aDataOut[119].0 := Diagnostics.b_EdmErrorSafetyShuntRelais;
OutProfinetSIEMENS.aDataOut[119].1 := Diagnostics.b_MeasurementIncomplete ;
OutProfinetSIEMENS.aDataOut[119].2 := Diagnostics.b_ValueOutOfRange;
OutProfinetSIEMENS.aDataOut[119].3 := Diagnostics.b_ExtControlCommFault;
OutProfinetSIEMENS.aDataOut[119].4 := Diagnostics.b_UPSLowVoltageWarning;
OutProfinetSIEMENS.aDataOut[119].5 := Diagnostics.b_UPSTimedShutdown;

OutProfinetSIEMENS.aDataOut[120].0 := OutProfinetSIEMENS.i_BessModeFB.0;
OutProfinetSIEMENS.aDataOut[120].1 := OutProfinetSIEMENS.i_BessModeFB.1;
OutProfinetSIEMENS.aDataOut[120].2 := OutProfinetSIEMENS.i_BessModeFB.2;
OutProfinetSIEMENS.aDataOut[120].3 := OutProfinetSIEMENS.i_InvModeFB.0;
OutProfinetSIEMENS.aDataOut[120].4 := OutProfinetSIEMENS.i_InvModeFB.1;

END_PROGRAM

// ---- POUs/ProfinetHandling/SiemensControl.TcPOU
PROGRAM SiemensControl
VAR
	r_CurrentLimMax						: REAL;
	r_CurrentLimMin						: REAL;
	fbRangeMinSoC : fbValueOutOfRange;
	fbRangeMaxSoC : fbValueOutOfRange;
	fbRangeVoltageDroop : fbValueOutOfRange;
	fbRangeFrequencyDroop : fbValueOutOfRange;
	fbRangeNomVoltage : fbValueOutOfRange;
	fbRangeNomFrequency : fbValueOutOfRange;
	fbRangeCurrentLimMax : fbValueOutOfRange;
	fbRangeCurrentLimMin : fbValueOutOfRange;
	fbRangeBaseCurrentRef : fbValueOutOfRange;
	fbRangeReactCurrentRef : fbValueOutOfRange;
	fbRangeRampRate : fbValueOutOfRange;
	
	w_TypeOfError								: WORD;
	b_TEST										: BOOL;
	
END_VAR

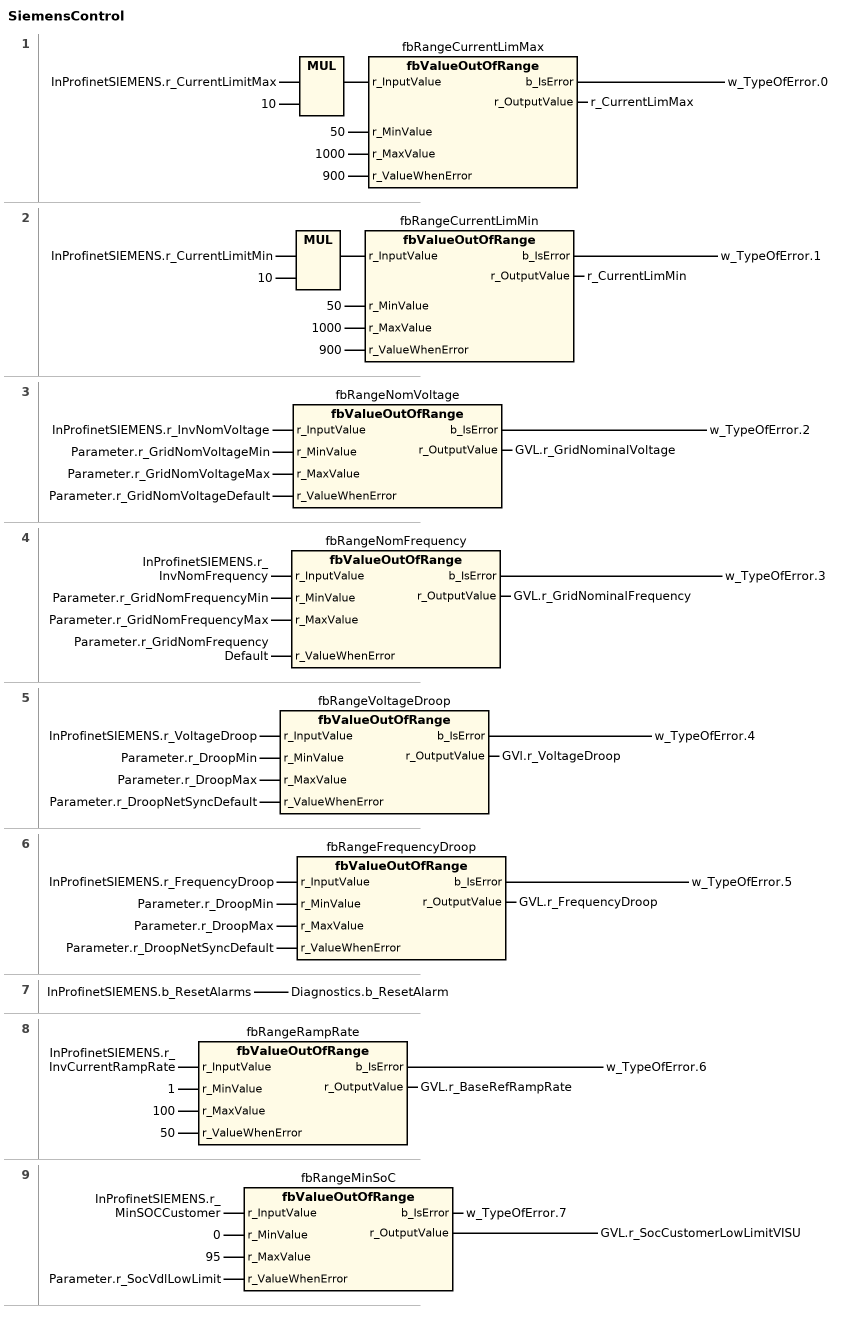
// NETWORK 1
fbRangeCurrentLimMax(
    r_InputValue := InProfinetSIEMENS.r_CurrentLimitMax * 10,
    r_MinValue := 50,
    r_MaxValue := 1000,
    r_ValueWhenError := 900,
    r_OutputValue => r_CurrentLimMax); // fbValueOutOfRange
w_TypeOfError.0 := fbRangeCurrentLimMax.b_IsError;

// NETWORK 2
fbRangeCurrentLimMin(
    r_InputValue := InProfinetSIEMENS.r_CurrentLimitMin * 10,
    r_MinValue := 50,
    r_MaxValue := 1000,
    r_ValueWhenError := 900,
    r_OutputValue => r_CurrentLimMin); // fbValueOutOfRange
w_TypeOfError.1 := fbRangeCurrentLimMin.b_IsError;

// NETWORK 3
fbRangeNomVoltage(
    r_InputValue := InProfinetSIEMENS.r_InvNomVoltage,
    r_MinValue := Parameter.r_GridNomVoltageMin,
    r_MaxValue := Parameter.r_GridNomVoltageMax,
    r_ValueWhenError := Parameter.r_GridNomVoltageDefault,
    r_OutputValue => GVL.r_GridNominalVoltage); // fbValueOutOfRange
w_TypeOfError.2 := fbRangeNomVoltage.b_IsError;

// NETWORK 4
fbRangeNomFrequency(
    r_InputValue := InProfinetSIEMENS.r_InvNomFrequency,
    r_MinValue := Parameter.r_GridNomFrequencyMin,
    r_MaxValue := Parameter.r_GridNomFrequencyMax,
    r_ValueWhenError := Parameter.r_GridNomFrequencyDefault,
    r_OutputValue => GVL.r_GridNominalFrequency); // fbValueOutOfRange
w_TypeOfError.3 := fbRangeNomFrequency.b_IsError;

// NETWORK 5
fbRangeVoltageDroop(
    r_InputValue := InProfinetSIEMENS.r_VoltageDroop,
    r_MinValue := Parameter.r_DroopMin,
    r_MaxValue := Parameter.r_DroopMax,
    r_ValueWhenError := Parameter.r_DroopNetSyncDefault,
    r_OutputValue => GVl.r_VoltageDroop); // fbValueOutOfRange
w_TypeOfError.4 := fbRangeVoltageDroop.b_IsError;

// NETWORK 6
fbRangeFrequencyDroop(
    r_InputValue := InProfinetSIEMENS.r_FrequencyDroop,
    r_MinValue := Parameter.r_DroopMin,
    r_MaxValue := Parameter.r_DroopMax,
    r_ValueWhenError := Parameter.r_DroopNetSyncDefault,
    r_OutputValue => GVL.r_FrequencyDroop); // fbValueOutOfRange
w_TypeOfError.5 := fbRangeFrequencyDroop.b_IsError;

// NETWORK 7
Diagnostics.b_ResetAlarm := InProfinetSIEMENS.b_ResetAlarms;

// NETWORK 8
fbRangeRampRate(
    r_InputValue := InProfinetSIEMENS.r_InvCurrentRampRate,
    r_MinValue := 1,
    r_MaxValue := 100,
    r_ValueWhenError := 50,
    r_OutputValue => GVL.r_BaseRefRampRate); // fbValueOutOfRange
w_TypeOfError.6 := fbRangeRampRate.b_IsError;

// NETWORK 9
fbRangeMinSoC(
    r_InputValue := InProfinetSIEMENS.r_MinSOCCustomer,
    r_MinValue := 0,
    r_MaxValue := 95,
    r_ValueWhenError := Parameter.r_SocVdlLowLimit,
    b_IsError => w_TypeOfError.7); // fbValueOutOfRange
GVL.r_SocCustomerLowLimitVISU := fbRangeMinSoC.r_OutputValue;

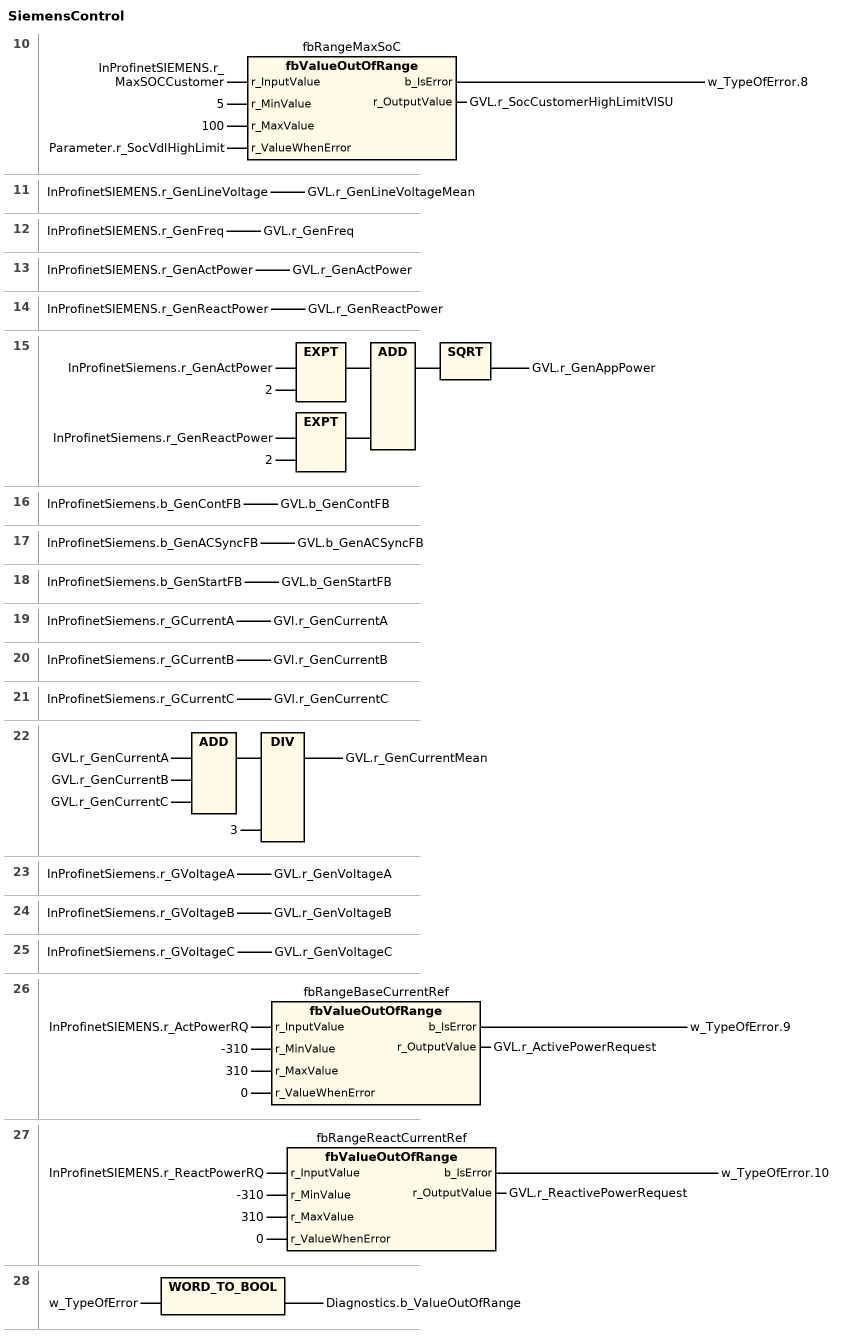
// NETWORK 10
fbRangeMaxSoC(
    r_InputValue := InProfinetSIEMENS.r_MaxSOCCustomer,
    r_MinValue := 5,
    r_MaxValue := 100,
    r_ValueWhenError := Parameter.r_SocVdlHighLimit,
    r_OutputValue => GVL.r_SocCustomerHighLimitVISU); // fbValueOutOfRange
w_TypeOfError.8 := fbRangeMaxSoC.b_IsError;

// NETWORK 11
GVL.r_GenLineVoltageMean := InProfinetSIEMENS.r_GenLineVoltage;

// NETWORK 12
GVL.r_GenFreq := InProfinetSIEMENS.r_GenFreq;

// NETWORK 13
GVL.r_GenActPower := InProfinetSIEMENS.r_GenActPower;

// NETWORK 14
GVL.r_GenReactPower := InProfinetSIEMENS.r_GenReactPower;

// NETWORK 15
GVL.r_GenAppPower := SQRT(EXPT(InProfinetSiemens.r_GenActPower, 2) + EXPT(InProfinetSiemens.r_GenReactPower, 2));

// NETWORK 16
GVL.b_GenContFB := InProfinetSiemens.b_GenContFB;

// NETWORK 17
GVL.b_GenACSyncFB := InProfinetSiemens.b_GenACSyncFB;

// NETWORK 18
GVL.b_GenStartFB := InProfinetSiemens.b_GenStartFB;

// NETWORK 19
GVl.r_GenCurrentA := InProfinetSiemens.r_GCurrentA;

// NETWORK 20
GVl.r_GenCurrentB := InProfinetSiemens.r_GCurrentB;

// NETWORK 21
GVl.r_GenCurrentC := InProfinetSiemens.r_GCurrentC;

// NETWORK 22
GVL.r_GenCurrentMean := (GVL.r_GenCurrentA + GVL.r_GenCurrentB + GVL.r_GenCurrentC) / 3;

// NETWORK 23
GVL.r_GenVoltageA := InProfinetSiemens.r_GVoltageA;

// NETWORK 24
GVL.r_GenVoltageB := InProfinetSiemens.r_GVoltageB;

// NETWORK 25
GVL.r_GenVoltageC := InProfinetSiemens.r_GVoltageC;

// NETWORK 26
fbRangeBaseCurrentRef(
    r_InputValue := InProfinetSIEMENS.r_ActPowerRQ,
    r_MinValue := -310,
    r_MaxValue := 310,
    r_ValueWhenError := 0,
    r_OutputValue => GVL.r_ActivePowerRequest); // fbValueOutOfRange
w_TypeOfError.9 := fbRangeBaseCurrentRef.b_IsError;

// NETWORK 27
fbRangeReactCurrentRef(
    r_InputValue := InProfinetSIEMENS.r_ReactPowerRQ,
    r_MinValue := -310,
    r_MaxValue := 310,
    r_ValueWhenError := 0,
    r_OutputValue => GVL.r_ReactivePowerRequest); // fbValueOutOfRange
w_TypeOfError.10 := fbRangeReactCurrentRef.b_IsError;

// NETWORK 28
Diagnostics.b_ValueOutOfRange := WORD_TO_BOOL(w_TypeOfError);

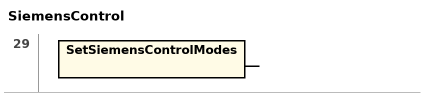
// NETWORK 29
SetSiemensControlModes();

END_PROGRAM
